(* IEC 61131-3 sources: OpenPLC_Sample_Programs/successed_ST, 85 files *)

(* ---- complex_arithmetic.st ---- *)
FUNCTION_BLOCK SLIDINGMEAN_A
  VAR_INPUT  START, END, VALUE : INT; END_VAR
  VAR MEAN : INT := 0; WEIGHT  : INT := 1; END_VAR
  VAR_OUTPUT Q : INT; END_VAR

  IF START < END THEN
    MEAN := (END - START) / WEIGHT * VALUE + MEAN;
    WEIGHT := END - START + WEIGHT;
  END_IF;
  Q := MEAN;
END_FUNCTION_BLOCK

FUNCTION_BLOCK SLIDINGMEAN_B
  VAR_INPUT  START, END, VALUE : INT;
             RESET : BOOL;
  END_VAR
  VAR MEAN :INT := 0; WEIGHT  : INT := 1; END_VAR
  VAR_OUTPUT Q : INT; END_VAR

  IF RESET THEN
    WEIGHT := 1; MEAN := 0;
  ELSIF START < END THEN
    MEAN := (END - START) * VALUE + WEIGHT * MEAN;
    WEIGHT := END - START + WEIGHT;
  END_IF;

END_FUNCTION_BLOCK

PROGRAM WARN_ABOVE
  VAR SENSOR, THRESHOLD : INT; END_VAR
  VAR SM : SLIDINGMEAN_A; END_VAR
  VAR_OUTPUT CRITICAL : BOOL; END_VAR
  SM(START := 0, END := 7, VALUE := SENSOR);
  CRITICAL :=  SM.Q > THRESHOLD;
END_PROGRAM

PROGRAM WARN_BELOW
  VAR SENSOR, THRESHOLD : INT; END_VAR
  VAR SM : SLIDINGMEAN_A; END_VAR
  VAR_OUTPUT CRITICAL : BOOL; END_VAR
  SM(START := 0, END := 7, VALUE := SENSOR);
  CRITICAL :=  SM.Q <= THRESHOLD;
END_PROGRAM

CONFIGURATION Config0
  RESOURCE Res0 ON PLC
    TASK TASK0(INTERVAL := T#50MS, PRIORITY := 0);
    PROGRAM INSTANCE0 WITH TASK0 : WARN_ABOVE;
    PROGRAM INSTANCE1 WITH TASK0 : WARN_BELOW;
  END_RESOURCE
END_CONFIGURATION

(* ---- fbembedding_1.st ---- *)
FUNCTION_BLOCK FB1

VAR_INPUT J : INT; END_VAR
VAR_OUTPUT P : INT; END_VAR
VAR SUM : INT; END_VAR

SUM := P + SUM;
P := SUM / P;

END_FUNCTION_BLOCK

PROGRAM MAIN
VAR_INPUT I : INT; END_VAR
VAR_OUTPUT O : INT; END_VAR

VAR
   A : FB1;
END_VAR
A(J:=I);
O:=A.P;
END_PROGRAM

CONFIGURATION Config0
  RESOURCE Res0 ON PLC
    TASK TASK0(INTERVAL := T#50MS, PRIORITY := 0);
    PROGRAM INSTANCE0 WITH TASK0 : MAIN;
  END_RESOURCE
END_CONFIGURATION

(* ---- lr.real.st ---- *)
TYPE
  OpMode : (Op , Teach);
  TeachStatus :  (Ok, NoTeachPoints, Teaching, InvalidTeachPoints, InvalidInputValue);
END_TYPE

FUNCTION_BLOCK TON_B

VAR_INPUT
  IN : BOOL;
  PT : INT;
END_VAR

VAR_OUTPUT
  Q  : BOOL;
  ET : INT;
END_VAR

IF IN THEN
  Q:= ET = INT#0;
  IF ET > INT#0 THEN
      ET := ET - INT#1;
  ELSE
      ET := INT#0;
  END_IF;
ELSE
  Q  := FALSE;
  ET := PT;
END_IF;

END_FUNCTION_BLOCK

PROGRAM Analogsensor

VAR
  SENSORINPUT_MIN : REAL := REAL#0.0;
  SENSORINPUT_MAX : REAL := REAL#4095.0;
  TEACHTIMEOUT : TIME := TIME#20s0ms;
END_VAR

VAR_INPUT
  TPSet : BOOL;
  SensorInput, TPy  : INT;
  OperationMode : OpMode;
END_VAR

VAR_OUTPUT
  SensorOutput : INT;
END_VAR

VAR
  initial          : BOOL;
  lastmode         : OpMode;
  Status           : TeachStatus;
  teachstep        : INT;
  x_temp, y_temp, t, m, x1, y1, x2, y2 : REAL;
  timeout          	: TON_B;
END_VAR

IF NOT initial THEN
  x1 := 0.0;
  y1 := 0.0;
  x2 := 0.0;
  y2 := 0.0;
  Status := TeachStatus#NoTeachPoints;
  initial := TRUE;
ELSE
  IF OperationMode = OpMode#Op THEN
    IF Status = TeachStatus#Ok AND INT_TO_REAL(SensorInput) >= SENSORINPUT_MIN AND INT_TO_REAL(SensorInput) <= SENSORINPUT_MAX THEN
      SensorOutput := REAL_TO_INT(m) * SensorInput + REAL_TO_INT(t);
    ELSE
      SensorOutput := 0;
    END_IF;
  ELSIF OperationMode = OpMode#Teach THEN
    IF lastmode <> OperationMode THEN
      teachstep := 0;
      timeout(IN := FALSE);
    END_IF;

    CASE teachstep OF
      0:
         Status := TeachStatus#Teaching;
         timeout(IN := TRUE, PT:=TIME_TO_INT(TEACHTIMEOUT));
         IF timeout.Q THEN
           OperationMode := OpMode#Op;
         END_IF;

         IF TPSet AND INT_TO_REAL(SensorInput) >= SENSORINPUT_MIN AND INT_TO_REAL(SensorInput) <= SENSORINPUT_MAX THEN
           y1 := INT_TO_REAL(TPy);
           x1 := INT_TO_REAL(SensorInput);
           teachstep := 1;
           timeout(IN := FALSE);
         END_IF;
      1:
         IF TPSet = FALSE THEN
           teachstep := 2;
         END_IF;
      2:
         timeout(IN := TRUE, PT:=TIME_TO_INT(TEACHTIMEOUT));

         IF timeout.Q THEN
           OperationMode := OpMode#Op;
         END_IF;

         IF TPSet AND INT_TO_REAL(SensorInput) >= SENSORINPUT_MIN
             AND INT_TO_REAL(SensorInput) <= SENSORINPUT_MAX THEN
           y2 := INT_TO_REAL(TPy);
           x2 := INT_TO_REAL(SensorInput);
           teachstep := 3;
           timeout(IN := FALSE);
         END_IF;
       3:
        IF x1 > x2 THEN
           x_temp := x1;
           y_temp := y1;
           x1 := x2;
           y1 := y2;
           x2 := x_temp;
           y2 := y_temp;
        END_IF;

        IF x2 - x1 <> 0.0 THEN
           m   := (y2 - y1) / (x2 - x1);
           t   := y1 - m * x1;
           Status := TeachStatus#Ok;
        ELSE
           Status := TeachStatus#InvalidTeachPoints;
           OperationMode := OpMode#Op;
         END_IF;
       END_CASE;
  END_IF;
END_IF;
  lastmode := OperationMode;
END_PROGRAM

CONFIGURATION Config0
  RESOURCE Res0 ON PLC
    TASK task0(INTERVAL := T#50ms, PRIORITY := 0);
    PROGRAM instance0 WITH task0 : Analogsensor;
  END_RESOURCE
END_CONFIGURATION

(* ---- PPU_13+ESystem.st ---- *)
(**********************************************************)
(* INCLUDED FROM ESYSTEM.ST                               *)

FUNCTION_BLOCK RS_FF
	VAR_INPUT    R,S : BOOL; END_VAR
	VAR_OUTPUT     Q : BOOL; END_VAR

	IF S THEN
		Q := TRUE;
	END_IF;
	IF R THEN
		Q := FALSE;
	END_IF;
END_FUNCTION_BLOCK

FUNCTION_BLOCK ESYSTEM
    VAR_INPUT RESET, MANUALSTAMPSLIDEROUT, MANUALSTAMPSLIDERIN,
    		    CRANEPRESSUREON,CRANEPRESSUREOFF: BOOL; END_VAR

    VAR_OUTPUT NEWCRANEPRESSURE : INT;
    			STAMPSLIDERIN, STAMPSLIDEROUT: BOOL; END_VAR

    VAR CONSTANT REGULARCRANEPRESSURE : INT := INT#8600; END_VAR

    VAR CRANEPRESSURE : RS_FF := (Q:=TRUE);
    	   RTRIGSTAMPSLIDERIN, RTRIGSTAMPSLIDEROUT : R_TRIG;
    END_VAR

	IF RESET THEN
		CRANEPRESSURE(S:=TRUE,R:=FALSE);
		RTRIGSTAMPSLIDERIN(CLK:=FALSE);
		RTRIGSTAMPSLIDEROUT(CLK:=FALSE);
	END_IF;

	CRANEPRESSURE(S:=CRANEPRESSUREON, R:=CRANEPRESSUREOFF);
	IF CRANEPRESSURE.Q THEN
		NEWCRANEPRESSURE := INT#0;
    	ELSE
    		NEWCRANEPRESSURE := REGULARCRANEPRESSURE;
    	END_IF;

	RTRIGSTAMPSLIDERIN(CLK:=STAMPSLIDERIN);
	RTRIGSTAMPSLIDEROUT(CLK:=STAMPSLIDEROUT);

	IF MANUALSTAMPSLIDEROUT AND RTRIGSTAMPSLIDERIN.Q THEN
		STAMPSLIDERIN := FALSE;
	ELSIF MANUALSTAMPSLIDEROUT THEN
		STAMPSLIDEROUT := TRUE;
	END_IF;

	IF MANUALSTAMPSLIDERIN AND RTRIGSTAMPSLIDEROUT.Q THEN
		STAMPSLIDEROUT := FALSE;
	ELSIF MANUALSTAMPSLIDEROUT THEN
		STAMPSLIDEROUT := TRUE;
	END_IF;
END_FUNCTION_BLOCK
(**********************************************************)

TYPE

    MAGAZIN_STATES_T : (GREEN_LAMP, INIT, INTERSTEP, MAGAZIN_INIT,
    MAGAZIN_INIT_2, SLIDER_MOVE_BACK, START_MAGAZIN, STEP0, STEP1, CONVEY);

    STAMP_STATES_T : (GREEN_LAMP, INIT, INTERSTEP, INTERSTEP_2, STAMPPROCESS,
    STAMPSLIDERBACK, STAMPSLIDERFORWARD, STAMP_INIT_1, STAMP_INIT_2,
    STAMP_INIT_3, STAMP_INIT_4, START_STAMP, STEP0, STEP1, STEP2);

    CRANE_STATES_T : (CRANE_GO_UP, CRANE_INIT, CRANE_INIT_2,
    CRANE_LIFT_AT_STAMP, CRANE_LIFT_CONVEYOR, CRANE_LIFT_CONVEYOR_BLACK,
    CRANE_LIFT_MAGAZIN, CRANE_LIFT_MAGAZIN_METALLIC,
    CRANE_LIFT_NOT_METALLIC_BLACK, CRANE_LOWER, CRANE_ON_CONVEYOR,
    CRANE_ON_CONVEYOR_METALLIC, CRANE_ON_CONVEYOR_NOT_METALLICA_BLACK,
    CRANE_ON_STAMP_METALLIC, CRANE_ON_STAMP_STOP_BLACK,
    CRANE_TURN_LEFT_BACK_TO_STAMP, CRANE_TURN_LEFT_FROM_STAMP,
    CRANE_TURN_LEFT_METALLIC, CRANE_TURN_LEFT_NOT_METALLIC,
    CRANE_TURN_LEFT_NOT_METALLIC_BLACK, INIT, INTERSTEP, INTERSTEP_2,
    LAST_WORKPIECE_AT_STAMP, LOWER_CRANE, MAGAZIN_STOP, MAGAZIN_STOP_BLACK,
    NO_WORKPIECE_READY, RESET_INTERCONNECT, START_CRANE, STEP0, SUCK_AT_STAMP,
    TIMEDELAY, TURN_RIGHT, TURN_RIGHT_BLACK, PAUSE, RELEASE, RELEASE_BLACK,
    RELEASE_WORKPIECE);

END_TYPE

FUNCTION_BLOCK MAGAZIN
    VAR_INPUT  CRANEDOWN : BOOL; END_VAR
    VAR_OUTPUT  CRANELOWER : BOOL; END_VAR
    VAR_INPUT  CRANEONCONVEYOR : BOOL; END_VAR
    VAR_INPUT  CRANEONMAGAZIN : BOOL; END_VAR
    VAR_INPUT  CRANESUCKED : BOOL; END_VAR
    VAR_OUTPUT  CRANETURNCLOCKWISE : BOOL; END_VAR
    VAR_OUTPUT  CRANETURNCOUNTERCLOCKWISE : BOOL; END_VAR
    VAR_INPUT  CRANEUP : BOOL; END_VAR
    VAR_OUTPUT  MAGAZINGREENLAMP : BOOL; END_VAR
    VAR_OUTPUT  MAGAZINSLIDER : BOOL; END_VAR
    VAR_OUTPUT  MAGAZINVACUUMOFF : BOOL; END_VAR
    VAR_OUTPUT  MAGAZINVACUUMON : BOOL; END_VAR
    VAR_OUTPUT  MAGAZINWHITELAMP : BOOL; END_VAR
    VAR  SFCINIT : BOOL; END_VAR
    VAR_INPUT  SFCRESET : BOOL; END_VAR
    VAR_INPUT  SLIDERMOVEDOUT : BOOL; END_VAR
    VAR_INPUT  SLIDERNOTMOVEDOUT : BOOL; END_VAR
    VAR_INPUT  STARTBUTTONMAGAZIN : BOOL; END_VAR
    VAR_OUTPUT  STARTCOMMANDMAGAZIN : BOOL; END_VAR
    VAR_INPUT  STARTVAR : BOOL; END_VAR
    VAR_INPUT  WORKPIECEREADY : BOOL; END_VAR
    VAR  _STATE : MAGAZIN_STATES_T; END_VAR
    VAR  _TRANSIT : BOOL; END_VAR
    VAR  INTERCONNECTMAGAZINSTARTCOMMAND : BOOL; END_VAR

    CASE _STATE OF
        MAGAZIN_STATES_T#GREEN_LAMP:
            _TRANSIT := FALSE;
            MAGAZINGREENLAMP := TRUE;
            INTERCONNECTMAGAZINSTARTCOMMAND := FALSE;
            IF TRUE THEN
                _TRANSIT := TRUE;
                _STATE := MAGAZIN_STATES_T#MAGAZIN_INIT;
            END_IF;

        MAGAZIN_STATES_T#INIT:
            _TRANSIT := FALSE;
            IF TRUE THEN
                _TRANSIT := TRUE;
                _STATE := MAGAZIN_STATES_T#START_MAGAZIN;
            END_IF;

        MAGAZIN_STATES_T#INTERSTEP:
            _TRANSIT := FALSE;
            STARTCOMMANDMAGAZIN := TRUE;
            IF STARTVAR THEN
                _TRANSIT := TRUE;
                _STATE := MAGAZIN_STATES_T#CONVEY;
            END_IF;

        MAGAZIN_STATES_T#MAGAZIN_INIT:
            _TRANSIT := FALSE;
            MAGAZINSLIDER := TRUE;
            IF TRUE THEN
                _TRANSIT := TRUE;
                _STATE := MAGAZIN_STATES_T#MAGAZIN_INIT_2;
            END_IF;

        MAGAZIN_STATES_T#MAGAZIN_INIT_2:
            _TRANSIT := FALSE;
            MAGAZINSLIDER := FALSE;
            IF TRUE THEN
                _TRANSIT := TRUE;
                _STATE := MAGAZIN_STATES_T#INTERSTEP;
            END_IF;

        MAGAZIN_STATES_T#SLIDER_MOVE_BACK:
            _TRANSIT := FALSE;
            IF ((SLIDERMOVEDOUT = TRUE) AND (SLIDERNOTMOVEDOUT = FALSE)) THEN
                MAGAZINSLIDER := FALSE;
            END_IF;
            IF CRANEUP THEN
                _TRANSIT := TRUE;
                _STATE := MAGAZIN_STATES_T#STEP1;
            END_IF;

        MAGAZIN_STATES_T#START_MAGAZIN:
            _TRANSIT := FALSE;
            MAGAZINSLIDER := FALSE;
            MAGAZINGREENLAMP := FALSE;
            STARTVAR := FALSE;
            STARTCOMMANDMAGAZIN := FALSE;
            IF (STARTBUTTONMAGAZIN = TRUE) THEN
                INTERCONNECTMAGAZINSTARTCOMMAND := TRUE;
            END_IF;
            IF INTERCONNECTMAGAZINSTARTCOMMAND THEN
                _TRANSIT := TRUE;
                _STATE := MAGAZIN_STATES_T#GREEN_LAMP;
            END_IF;

        MAGAZIN_STATES_T#STEP0:
            _TRANSIT := FALSE;
            IF CRANEDOWN THEN
                _TRANSIT := TRUE;
                _STATE := MAGAZIN_STATES_T#SLIDER_MOVE_BACK;
            END_IF;

        MAGAZIN_STATES_T#STEP1:
            _TRANSIT := FALSE;
            IF CRANEONCONVEYOR THEN
                _TRANSIT := TRUE;
                _STATE := MAGAZIN_STATES_T#INTERSTEP;
            END_IF;

        MAGAZIN_STATES_T#CONVEY:
            _TRANSIT := FALSE;
            IF SLIDERNOTMOVEDOUT THEN
                MAGAZINSLIDER := TRUE;
            END_IF;
            IF CRANEONMAGAZIN THEN
                _TRANSIT := TRUE;
                _STATE := MAGAZIN_STATES_T#STEP0;
            END_IF;

            END_CASE;
END_FUNCTION_BLOCK

FUNCTION_BLOCK STAMP_FB
VAR_INPUT  CRANEDOWN : BOOL; END_VAR
VAR_INPUT  CRANEONCONVEYOR : BOOL; END_VAR
VAR_INPUT  CRANEPOSITIONSTAMP : BOOL; END_VAR
VAR_INPUT  CRANESUCKED : BOOL; END_VAR
VAR_INPUT  CRANEUP : BOOL; END_VAR
VAR  DURATION : TIME := TIME#500MS; END_VAR
VAR  SFCINIT : BOOL; END_VAR
VAR_INPUT  SFCRESET : BOOL; END_VAR
VAR_OUTPUT  STAMPGREENLAMP : BOOL; END_VAR
VAR_INPUT  STAMPLOWERED : BOOL; END_VAR
VAR_OUTPUT  STAMPPRESSURE : BOOL; END_VAR
VAR_OUTPUT  STAMPPUSHER : BOOL; END_VAR
VAR_INPUT  STAMPSLIDERFILLED : BOOL; END_VAR
VAR_OUTPUT  STAMPSLIDERMOVEDIN : BOOL; END_VAR
VAR_OUTPUT  STAMPSLIDERMOVEDOUT : BOOL; END_VAR
VAR_INPUT  STAMPSLIDERSENSORMOVEDIN : BOOL; END_VAR
VAR_INPUT  STAMPSLIDERSENSORMOVEDOUT : BOOL; END_VAR
VAR_INPUT  STAMPSTARTBUTTON : BOOL; END_VAR
VAR_INPUT  STAMPUP : BOOL; END_VAR
VAR_OUTPUT  STAMPWHITELAMP : BOOL; END_VAR
VAR_OUTPUT  STARTCOMMANDSTAMP : BOOL; END_VAR
VAR_INPUT  STARTVAR : BOOL; END_VAR
VAR  TIMER : TON; END_VAR
VAR  _STATE : STAMP_STATES_T; END_VAR
VAR  _TRANSIT : BOOL; END_VAR
VAR  INTERCONNECT : BOOL; END_VAR
VAR  INTERCONNECTSTAMPSTARTCOMMAND : BOOL; END_VAR

CASE _STATE OF
    STAMP_STATES_T#GREEN_LAMP:
        _TRANSIT := FALSE;
        STAMPGREENLAMP := TRUE;
        INTERCONNECTSTAMPSTARTCOMMAND := FALSE;
        IF TRUE THEN
            _TRANSIT := TRUE;
            _STATE := STAMP_STATES_T#STAMP_INIT_1;
        END_IF;

    STAMP_STATES_T#INIT:
        _TRANSIT := FALSE;
        IF TRUE THEN
            _TRANSIT := TRUE;
            _STATE := STAMP_STATES_T#START_STAMP;
        END_IF;

    STAMP_STATES_T#INTERSTEP:
        _TRANSIT := FALSE;
        STARTCOMMANDSTAMP := TRUE;
        IF STARTVAR THEN
            _TRANSIT := TRUE;
            _STATE := STAMP_STATES_T#INTERSTEP_2;
        END_IF;

    STAMP_STATES_T#INTERSTEP_2:
        _TRANSIT := FALSE;
        IF STAMPSLIDERFILLED THEN
            _TRANSIT := TRUE;
            _STATE := STAMP_STATES_T#STEP0;
        END_IF;

    STAMP_STATES_T#STAMPPROCESS:
        _TRANSIT := FALSE;
        STAMPSLIDERMOVEDIN := FALSE;
        STAMPPUSHER := TRUE;
        IF STAMPLOWERED THEN
            _TRANSIT := TRUE;
            _STATE := STAMP_STATES_T#STEP1;
        END_IF;

    STAMP_STATES_T#STAMPSLIDERBACK:
        _TRANSIT := FALSE;
        STAMPSLIDERMOVEDIN := TRUE;
        STAMPSLIDERMOVEDOUT := FALSE;
        IF STAMPSLIDERSENSORMOVEDIN THEN
            _TRANSIT := TRUE;
            _STATE := STAMP_STATES_T#STAMPPROCESS;
        END_IF;

    STAMP_STATES_T#STAMPSLIDERFORWARD:
        _TRANSIT := FALSE;
        STAMPPUSHER := FALSE;
        STAMPSLIDERMOVEDOUT := TRUE;
        IF ((STAMPLOWERED = FALSE) AND (STAMPUP = TRUE)) THEN
            INTERCONNECT := FALSE;
        END_IF;
        TIMER(IN := FALSE, PT := TIME#1MS);
        IF STAMPSLIDERMOVEDOUT THEN
            _TRANSIT := TRUE;
            _STATE := STAMP_STATES_T#STEP2;
        END_IF;

    STAMP_STATES_T#STAMP_INIT_1:
        _TRANSIT := FALSE;
        STAMPSLIDERMOVEDIN := TRUE;
        STAMPSLIDERMOVEDOUT := FALSE;
        IF STAMPSLIDERSENSORMOVEDIN THEN
            _TRANSIT := TRUE;
            _STATE := STAMP_STATES_T#STAMP_INIT_2;
        END_IF;

    STAMP_STATES_T#STAMP_INIT_2:
        _TRANSIT := FALSE;
        STAMPSLIDERMOVEDIN := FALSE;
        STAMPSLIDERMOVEDOUT := TRUE;
        IF STAMPSLIDERSENSORMOVEDOUT THEN
            _TRANSIT := TRUE;
            _STATE := STAMP_STATES_T#STAMP_INIT_3;
        END_IF;

    STAMP_STATES_T#STAMP_INIT_3:
        _TRANSIT := FALSE;
        STAMPPUSHER := TRUE;
        IF STAMPLOWERED THEN
            _TRANSIT := TRUE;
            _STATE := STAMP_STATES_T#STAMP_INIT_4;
        END_IF;

    STAMP_STATES_T#STAMP_INIT_4:
        _TRANSIT := FALSE;
        STAMPPUSHER := FALSE;
        IF STAMPUP THEN
            _TRANSIT := TRUE;
            _STATE := STAMP_STATES_T#INTERSTEP;
        END_IF;

    STAMP_STATES_T#START_STAMP:
        _TRANSIT := FALSE;
        STAMPSLIDERMOVEDOUT := FALSE;
        STAMPSLIDERMOVEDIN := FALSE;
        STAMPPUSHER := FALSE;
        STAMPGREENLAMP := FALSE;
        STAMPPRESSURE := FALSE;
        STARTCOMMANDSTAMP := FALSE;
        IF (STAMPSTARTBUTTON = TRUE) THEN
            INTERCONNECTSTAMPSTARTCOMMAND := TRUE;
        END_IF;
        IF INTERCONNECTSTAMPSTARTCOMMAND THEN
            _TRANSIT := TRUE;
            _STATE := STAMP_STATES_T#GREEN_LAMP;
        END_IF;

    STAMP_STATES_T#STEP0:
        _TRANSIT := FALSE;
        IF CRANEUP THEN
            _TRANSIT := TRUE;
            _STATE := STAMP_STATES_T#STAMPSLIDERBACK;
        END_IF;

    STAMP_STATES_T#STEP1:
        _TRANSIT := FALSE;
        TIMER(IN := STAMPLOWERED, PT := TIME#12MS);
        INTERCONNECT := TIMER.Q;
        IF INTERCONNECT THEN
            _TRANSIT := TRUE;
            _STATE := STAMP_STATES_T#STAMPSLIDERFORWARD;
        END_IF;

    STAMP_STATES_T#STEP2:
        _TRANSIT := FALSE;
        IF (CRANEONCONVEYOR AND NOT STAMPSLIDERFILLED) THEN
            _TRANSIT := TRUE;
            _STATE := STAMP_STATES_T#INTERSTEP;
        END_IF;

    END_CASE;
END_FUNCTION_BLOCK

FUNCTION_BLOCK CRANE_FB
VAR  CRANTURNCLOCKWISE : BOOL; END_VAR
VAR_INPUT  CRANEDOWN : BOOL; END_VAR
VAR_OUTPUT  CRANELOWER : BOOL; END_VAR
VAR_INPUT  CRANEONCONVEYOR : BOOL; END_VAR
VAR_INPUT  CRANEONMAGAZIN : BOOL; END_VAR
VAR_INPUT  CRANEPOSITIONSTAMP : BOOL; END_VAR
VAR_INPUT  CRANESUCKED : BOOL; END_VAR
VAR_OUTPUT  CRANETURNCLOCKWISE : BOOL; END_VAR
VAR_OUTPUT  CRANETURNCOUNTERCLOCKWISE : BOOL; END_VAR
VAR_INPUT  CRANEUP : BOOL; END_VAR
VAR  DURATION1 : TIME := TIME#1S500MS; END_VAR
VAR_INPUT  MAGAZINCAPACITIVESENSOR : BOOL; END_VAR
VAR_OUTPUT  MAGAZINSLIDER : BOOL; END_VAR
VAR_OUTPUT  MAGAZINVACUUMOFF : BOOL; END_VAR
VAR_OUTPUT  MAGAZINVACUUMON : BOOL; END_VAR
VAR  SFCINIT : BOOL; END_VAR
VAR_INPUT  SFCRESET : BOOL; END_VAR
VAR_INPUT  SLIDERMOVEDOUT : BOOL; END_VAR
VAR_INPUT  SLIDERNOTMOVEDOUT : BOOL; END_VAR
VAR_INPUT  STAMPLOWERED : BOOL; END_VAR
VAR_INPUT  STAMPSLIDERFILLED : BOOL; END_VAR
VAR_INPUT  STARTBUTTONMAGAZIN : BOOL; END_VAR
VAR_OUTPUT  STARTCOMMANDCRANE : BOOL; END_VAR
VAR_INPUT  STARTVAR : BOOL; END_VAR
VAR  TIMEDELAY_TIMER : TON; END_VAR
VAR  TIMEDELAY_TIMER_DURATION : TIME := TIME#50MS; END_VAR
VAR  TIMEDELAY_TIMER_INTERCONNECT : BOOL; END_VAR
VAR  TIMER1 : TON; END_VAR
VAR_INPUT  WORKPIECEREADY : BOOL; END_VAR
VAR  _STATE : CRANE_STATES_T; END_VAR
VAR  _TRANSIT : BOOL; END_VAR
VAR  ACTUALTIME1 : TIME; END_VAR
VAR  INTERCONNECT : BOOL; END_VAR
VAR  INTERCONNECTCRANESTARTCOMMAND : BOOL; END_VAR

CASE _STATE OF
    CRANE_STATES_T#CRANE_GO_UP:
        _TRANSIT := FALSE;
        CRANELOWER := FALSE;
        IF (CRANEUP AND (MAGAZINCAPACITIVESENSOR OR NOT WORKPIECEREADY)) THEN
            _TRANSIT := TRUE;
            _STATE := CRANE_STATES_T#PAUSE;
        ELSIF ((CRANEUP AND NOT MAGAZINCAPACITIVESENSOR) AND WORKPIECEREADY) THEN
            _TRANSIT := TRUE;
            _STATE := CRANE_STATES_T#TURN_RIGHT_BLACK;
        END_IF;

    CRANE_STATES_T#CRANE_INIT:
        _TRANSIT := FALSE;
        CRANELOWER := TRUE;
        INTERCONNECTCRANESTARTCOMMAND := FALSE;
        IF CRANEDOWN THEN
            _TRANSIT := TRUE;
            _STATE := CRANE_STATES_T#CRANE_INIT_2;
        END_IF;

    CRANE_STATES_T#CRANE_INIT_2:
        _TRANSIT := FALSE;
        CRANELOWER := FALSE;
        IF CRANEUP THEN
            _TRANSIT := TRUE;
            _STATE := CRANE_STATES_T#INTERSTEP;
        END_IF;

    CRANE_STATES_T#CRANE_LIFT_AT_STAMP:
        _TRANSIT := FALSE;
        CRANELOWER := FALSE;
        IF CRANEUP THEN
            _TRANSIT := TRUE;
            _STATE := CRANE_STATES_T#CRANE_TURN_LEFT_FROM_STAMP;
        END_IF;

    CRANE_STATES_T#CRANE_LIFT_CONVEYOR:
        _TRANSIT := FALSE;
        CRANELOWER := FALSE;
        IF TRUE THEN
            _TRANSIT := TRUE;
            _STATE := CRANE_STATES_T#INTERSTEP;
        END_IF;

    CRANE_STATES_T#CRANE_LIFT_CONVEYOR_BLACK:
        _TRANSIT := FALSE;
        CRANELOWER := FALSE;
        IF CRANEUP THEN
            _TRANSIT := TRUE;
            _STATE := CRANE_STATES_T#CRANE_TURN_LEFT_BACK_TO_STAMP;
        END_IF;

    CRANE_STATES_T#CRANE_LIFT_MAGAZIN:
        _TRANSIT := FALSE;
        CRANELOWER := FALSE;
        IF CRANEUP THEN
            _TRANSIT := TRUE;
            _STATE := CRANE_STATES_T#CRANE_TURN_LEFT_NOT_METALLIC;
        END_IF;

    CRANE_STATES_T#CRANE_LIFT_MAGAZIN_METALLIC:
        _TRANSIT := FALSE;
        CRANELOWER := FALSE;
        IF CRANEUP THEN
            _TRANSIT := TRUE;
            _STATE := CRANE_STATES_T#CRANE_TURN_LEFT_METALLIC;
        END_IF;

    CRANE_STATES_T#CRANE_LIFT_NOT_METALLIC_BLACK:
        _TRANSIT := FALSE;
        CRANELOWER := FALSE;
        IF CRANEUP THEN
            _TRANSIT := TRUE;
            _STATE := CRANE_STATES_T#CRANE_TURN_LEFT_NOT_METALLIC_BLACK;
        END_IF;

    CRANE_STATES_T#CRANE_LOWER:
        _TRANSIT := FALSE;
        MAGAZINVACUUMON := TRUE;
        MAGAZINVACUUMOFF := FALSE;
        CRANELOWER := TRUE;
        IF CRANESUCKED THEN
            _TRANSIT := TRUE;
            _STATE := CRANE_STATES_T#STEP0;
        END_IF;

    CRANE_STATES_T#CRANE_ON_CONVEYOR:
        _TRANSIT := FALSE;
        CRANETURNCOUNTERCLOCKWISE := FALSE;
        CRANETURNCLOCKWISE := FALSE;
        CRANELOWER := TRUE;
        IF CRANEDOWN THEN
            _TRANSIT := TRUE;
            _STATE := CRANE_STATES_T#RELEASE;
        END_IF;

    CRANE_STATES_T#CRANE_ON_CONVEYOR_METALLIC:
        _TRANSIT := FALSE;
        CRANETURNCOUNTERCLOCKWISE := FALSE;
        CRANETURNCLOCKWISE := FALSE;
        CRANELOWER := TRUE;
        IF CRANEDOWN THEN
            _TRANSIT := TRUE;
            _STATE := CRANE_STATES_T#RELEASE;
        END_IF;

    CRANE_STATES_T#CRANE_ON_CONVEYOR_NOT_METALLICA_BLACK:
        _TRANSIT := FALSE;
        CRANETURNCOUNTERCLOCKWISE := FALSE;
        CRANETURNCLOCKWISE := FALSE;
        CRANELOWER := TRUE;
        IF CRANEDOWN THEN
            _TRANSIT := TRUE;
            _STATE := CRANE_STATES_T#RELEASE_BLACK;
        END_IF;

    CRANE_STATES_T#CRANE_ON_STAMP_METALLIC:
        _TRANSIT := FALSE;
        CRANETURNCOUNTERCLOCKWISE := FALSE;
        CRANETURNCLOCKWISE := FALSE;
        CRANELOWER := TRUE;
        IF CRANEDOWN THEN
            _TRANSIT := TRUE;
            _STATE := CRANE_STATES_T#RELEASE_WORKPIECE;
        END_IF;

    CRANE_STATES_T#CRANE_ON_STAMP_STOP_BLACK:
        _TRANSIT := FALSE;
        CRANETURNCLOCKWISE := FALSE;
        CRANETURNCOUNTERCLOCKWISE := FALSE;
        IF TRUE THEN
            _TRANSIT := TRUE;
            _STATE := CRANE_STATES_T#RESET_INTERCONNECT;
        END_IF;

    CRANE_STATES_T#CRANE_TURN_LEFT_BACK_TO_STAMP:
        _TRANSIT := FALSE;
        CRANETURNCOUNTERCLOCKWISE := TRUE;
        CRANETURNCLOCKWISE := FALSE;
        IF CRANEPOSITIONSTAMP THEN
            _TRANSIT := TRUE;
            _STATE := CRANE_STATES_T#CRANE_ON_STAMP_STOP_BLACK;
        END_IF;

    CRANE_STATES_T#CRANE_TURN_LEFT_FROM_STAMP:
        _TRANSIT := FALSE;
        CRANETURNCLOCKWISE := TRUE;
        CRANETURNCOUNTERCLOCKWISE := FALSE;
        IF CRANEONCONVEYOR THEN
            _TRANSIT := TRUE;
            _STATE := CRANE_STATES_T#CRANE_ON_CONVEYOR_METALLIC;
        END_IF;

    CRANE_STATES_T#CRANE_TURN_LEFT_METALLIC:
        _TRANSIT := FALSE;
        CRANETURNCOUNTERCLOCKWISE := TRUE;
        CRANETURNCLOCKWISE := FALSE;
        IF CRANEPOSITIONSTAMP THEN
            _TRANSIT := TRUE;
            _STATE := CRANE_STATES_T#CRANE_ON_STAMP_METALLIC;
        END_IF;

    CRANE_STATES_T#CRANE_TURN_LEFT_NOT_METALLIC:
        _TRANSIT := FALSE;
        CRANETURNCOUNTERCLOCKWISE := TRUE;
        CRANETURNCLOCKWISE := FALSE;
        IF CRANEONCONVEYOR THEN
            _TRANSIT := TRUE;
            _STATE := CRANE_STATES_T#CRANE_ON_CONVEYOR;
        END_IF;

    CRANE_STATES_T#CRANE_TURN_LEFT_NOT_METALLIC_BLACK:
        _TRANSIT := FALSE;
        CRANETURNCOUNTERCLOCKWISE := TRUE;
        CRANETURNCLOCKWISE := FALSE;
        IF CRANEONCONVEYOR THEN
            _TRANSIT := TRUE;
            _STATE := CRANE_STATES_T#CRANE_ON_CONVEYOR_NOT_METALLICA_BLACK;
        END_IF;

    CRANE_STATES_T#INIT:
        _TRANSIT := FALSE;
        IF TRUE THEN
            _TRANSIT := TRUE;
            _STATE := CRANE_STATES_T#START_CRANE;
        END_IF;

    CRANE_STATES_T#INTERSTEP:
        _TRANSIT := FALSE;
        STARTCOMMANDCRANE := TRUE;
        IF STARTVAR THEN
            _TRANSIT := TRUE;
            _STATE := CRANE_STATES_T#INTERSTEP_2;
        END_IF;

    CRANE_STATES_T#INTERSTEP_2:
        _TRANSIT := FALSE;
        IF SLIDERMOVEDOUT THEN
            _TRANSIT := TRUE;
            _STATE := CRANE_STATES_T#TIMEDELAY;
        END_IF;

    CRANE_STATES_T#LAST_WORKPIECE_AT_STAMP:
        _TRANSIT := FALSE;
        IF TRUE THEN
            _TRANSIT := TRUE;
            _STATE := CRANE_STATES_T#PAUSE;
        END_IF;

    CRANE_STATES_T#LOWER_CRANE:
        _TRANSIT := FALSE;
        CRANELOWER := TRUE;
        IF CRANEDOWN THEN
            _TRANSIT := TRUE;
            _STATE := CRANE_STATES_T#SUCK_AT_STAMP;
        END_IF;

    CRANE_STATES_T#MAGAZIN_STOP:
        _TRANSIT := FALSE;
        CRANETURNCLOCKWISE := FALSE;
        CRANETURNCOUNTERCLOCKWISE := FALSE;
        IF (NOT WORKPIECEREADY AND NOT STAMPSLIDERFILLED) THEN
            _TRANSIT := TRUE;
            _STATE := CRANE_STATES_T#NO_WORKPIECE_READY;
        ELSIF WORKPIECEREADY THEN
            _TRANSIT := TRUE;
            _STATE := CRANE_STATES_T#CRANE_LOWER;
        ELSIF (NOT WORKPIECEREADY AND STAMPSLIDERFILLED) THEN
            _TRANSIT := TRUE;
            _STATE := CRANE_STATES_T#LAST_WORKPIECE_AT_STAMP;
        END_IF;

    CRANE_STATES_T#MAGAZIN_STOP_BLACK:
        _TRANSIT := FALSE;
        CRANETURNCLOCKWISE := FALSE;
        CRANETURNCOUNTERCLOCKWISE := FALSE;
        MAGAZINVACUUMON := TRUE;
        MAGAZINVACUUMOFF := FALSE;
        CRANELOWER := TRUE;
        IF CRANESUCKED THEN
            _TRANSIT := TRUE;
            _STATE := CRANE_STATES_T#CRANE_LIFT_NOT_METALLIC_BLACK;
        END_IF;

    CRANE_STATES_T#NO_WORKPIECE_READY:
        _TRANSIT := FALSE;
        IF TRUE THEN
            _TRANSIT := TRUE;
            _STATE := CRANE_STATES_T#START_CRANE;
        END_IF;

    CRANE_STATES_T#RESET_INTERCONNECT:
        _TRANSIT := FALSE;
        INTERCONNECT := FALSE;
        TIMER1(IN := FALSE, PT := TIME#1MS);
        IF SLIDERMOVEDOUT THEN
            _TRANSIT := TRUE;
            _STATE := CRANE_STATES_T#LOWER_CRANE;
        END_IF;

    CRANE_STATES_T#START_CRANE:
        _TRANSIT := FALSE;
        CRANELOWER := FALSE;
        MAGAZINVACUUMOFF := TRUE;
        MAGAZINVACUUMON := FALSE;
        CRANETURNCOUNTERCLOCKWISE := FALSE;
        CRANETURNCLOCKWISE := FALSE;
        STARTVAR := FALSE;
        STARTCOMMANDCRANE := FALSE;
        IF (STARTBUTTONMAGAZIN = TRUE) THEN
            INTERCONNECTCRANESTARTCOMMAND := TRUE;
        END_IF;
        IF INTERCONNECTCRANESTARTCOMMAND THEN
            _TRANSIT := TRUE;
            _STATE := CRANE_STATES_T#CRANE_INIT;
        END_IF;

    CRANE_STATES_T#STEP0:
        _TRANSIT := FALSE;
        IF NOT MAGAZINCAPACITIVESENSOR THEN
            _TRANSIT := TRUE;
            _STATE := CRANE_STATES_T#CRANE_LIFT_MAGAZIN;
        ELSIF MAGAZINCAPACITIVESENSOR THEN
            _TRANSIT := TRUE;
            _STATE := CRANE_STATES_T#CRANE_LIFT_MAGAZIN_METALLIC;
        END_IF;

    CRANE_STATES_T#SUCK_AT_STAMP:
        _TRANSIT := FALSE;
        MAGAZINVACUUMON := TRUE;
        MAGAZINVACUUMOFF := FALSE;
        IF CRANESUCKED THEN
            _TRANSIT := TRUE;
            _STATE := CRANE_STATES_T#CRANE_LIFT_AT_STAMP;
        END_IF;

    CRANE_STATES_T#TIMEDELAY:
        _TRANSIT := FALSE;
        TIMEDELAY_TIMER(IN := TRUE, PT := TIMEDELAY_TIMER_DURATION);
        TIMEDELAY_TIMER_INTERCONNECT := TIMEDELAY_TIMER.Q;
        IF TIMEDELAY_TIMER_INTERCONNECT THEN
            _TRANSIT := TRUE;
            _STATE := CRANE_STATES_T#TURN_RIGHT;
        END_IF;

    CRANE_STATES_T#TURN_RIGHT:
        _TRANSIT := FALSE;
        CRANETURNCLOCKWISE := TRUE;
        CRANETURNCOUNTERCLOCKWISE := FALSE;
        IF CRANEONMAGAZIN THEN
            _TRANSIT := TRUE;
            _STATE := CRANE_STATES_T#MAGAZIN_STOP;
        END_IF;

    CRANE_STATES_T#TURN_RIGHT_BLACK:
        _TRANSIT := FALSE;
        CRANETURNCLOCKWISE := TRUE;
        CRANETURNCOUNTERCLOCKWISE := FALSE;
        IF CRANEONMAGAZIN THEN
            _TRANSIT := TRUE;
            _STATE := CRANE_STATES_T#MAGAZIN_STOP_BLACK;
        END_IF;

    CRANE_STATES_T#PAUSE:
        _TRANSIT := FALSE;
        TIMER1(IN := CRANEUP, PT := DURATION1);
        INTERCONNECT := TIMER1.Q;
        IF INTERCONNECT THEN
            _TRANSIT := TRUE;
            _STATE := CRANE_STATES_T#RESET_INTERCONNECT;
        END_IF;

    CRANE_STATES_T#RELEASE:
        _TRANSIT := FALSE;
        MAGAZINVACUUMOFF := TRUE;
        MAGAZINVACUUMON := FALSE;
        IF TRUE THEN
            _TRANSIT := TRUE;
            _STATE := CRANE_STATES_T#CRANE_LIFT_CONVEYOR;
        END_IF;

    CRANE_STATES_T#RELEASE_BLACK:
        _TRANSIT := FALSE;
        MAGAZINVACUUMON := FALSE;
        MAGAZINVACUUMOFF := TRUE;
        IF TRUE THEN
            _TRANSIT := TRUE;
            _STATE := CRANE_STATES_T#CRANE_LIFT_CONVEYOR_BLACK;
        END_IF;

    CRANE_STATES_T#RELEASE_WORKPIECE:
        _TRANSIT := FALSE;
        MAGAZINVACUUMOFF := TRUE;
        MAGAZINVACUUMON := FALSE;
        IF TRUE THEN
            _TRANSIT := TRUE;
            _STATE := CRANE_STATES_T#CRANE_GO_UP;
        END_IF;

    END_CASE;
END_FUNCTION_BLOCK

PROGRAM MAIN

        (** NEW VARIABLES **)
	VAR EMERGENCY : ESYSTEM; END_VAR
	VAR_INPUT
	    SENSOR_MANUALSTAMPSLIDEROUT, SENSOR_MANUALSTAMPSLIDERIN,
	    SENSOR_CRANEPRESSUREON, SENSOR_CRANEPRESSUREOFF : BOOL;
	END_VAR

VAR  CRANE : CRANE_FB; END_VAR
VAR  MAG : MAGAZIN; END_VAR

VAR_OUTPUT ACTUATOR_ANALOGCRANEPRESSURE : INT; END_VAR
VAR_OUTPUT ACTUATOR_CRANELOWER : BOOL; END_VAR
VAR_OUTPUT ACTUATOR_CRANETURNCLOCKWISE : BOOL; END_VAR
VAR_OUTPUT ACTUATOR_CRANETURNCOUNTERCLOCKWISE : BOOL; END_VAR
VAR_OUTPUT ACTUATOR_MAGAZINGREENLAMP : BOOL; END_VAR
VAR_OUTPUT ACTUATOR_MAGAZINSLIDER : BOOL; END_VAR
VAR_OUTPUT ACTUATOR_MAGAZINVACUUMOFF : BOOL; END_VAR
VAR_OUTPUT ACTUATOR_MAGAZINVACUUMON : BOOL; END_VAR
VAR_OUTPUT ACTUATOR_MAGAZINWHITELAMP : BOOL; END_VAR
VAR_OUTPUT ACTUATOR_STAMPGREENLAMP : BOOL; END_VAR
VAR_OUTPUT ACTUATOR_STAMPPUSHER : BOOL; END_VAR
VAR_OUTPUT ACTUATOR_STAMPSLIDERMOVEDIN : BOOL; END_VAR
VAR_OUTPUT ACTUATOR_STAMPSLIDERMOVEDOUT : BOOL; END_VAR
VAR_OUTPUT ACTUATOR_STAMPWHITELAMP : BOOL; END_VAR
VAR_INPUT SENSOR_CRANEDOWN : BOOL; END_VAR
VAR_INPUT SENSOR_CRANEONCONVEYOR : BOOL; END_VAR
VAR_INPUT SENSOR_CRANEONMAGAZIN : BOOL; END_VAR
VAR_INPUT SENSOR_CRANEPOSITION : BOOL; END_VAR
VAR_INPUT SENSOR_CRANEPOSITIONSTAMP : BOOL; END_VAR
VAR_INPUT SENSOR_CRANESUCKED : BOOL; END_VAR
VAR_INPUT SENSOR_CRANEUP : BOOL; END_VAR
VAR_INPUT SENSOR_MAGAZINCAPACITIVESENSOR : BOOL; END_VAR
VAR_INPUT SENSOR_MAGAZINEMERGENCYSTOP : BOOL; END_VAR
VAR_INPUT SENSOR_MAGAZINOPTICALSENSOR : BOOL; END_VAR
VAR_INPUT SENSOR_MAGAZINSWITCHMANUELLAUTOMATIC : BOOL; END_VAR
VAR_INPUT SENSOR_SLIDERMOVEDOUT : BOOL; END_VAR
VAR_INPUT SENSOR_SLIDERNOTMOVEDOUT : BOOL; END_VAR
VAR_INPUT SENSOR_STAMPEMERGENCYSTOP : BOOL; END_VAR
VAR_INPUT SENSOR_STAMPLOWERED : BOOL; END_VAR
VAR_INPUT SENSOR_STAMPSLIDERFILLED : BOOL; END_VAR
VAR_INPUT SENSOR_STAMPSLIDERSENSORMOVEDIN : BOOL; END_VAR
VAR_INPUT SENSOR_STAMPSLIDERSENSORMOVEDOUT : BOOL; END_VAR
VAR_INPUT SENSOR_STAMPSTARTBUTTON : BOOL; END_VAR
VAR_INPUT SENSOR_STAMPSWITCHMANUELLAUTOMATIC : BOOL; END_VAR
VAR_INPUT SENSOR_STAMPUP : BOOL; END_VAR
VAR_INPUT SENSOR_STARTBUTTONMAGAZIN : BOOL; END_VAR
VAR_INPUT SENSOR_WORKPIECEREADY : BOOL; END_VAR
VAR  STAMP : STAMP_FB; END_VAR

CRANE.CRANEDOWN := SENSOR_CRANEDOWN;
CRANE.CRANEONCONVEYOR := SENSOR_CRANEONCONVEYOR;
CRANE.CRANEONMAGAZIN := SENSOR_CRANEONMAGAZIN;
CRANE.CRANEPOSITIONSTAMP := SENSOR_CRANEPOSITIONSTAMP;
CRANE.CRANESUCKED := SENSOR_CRANESUCKED;
CRANE.CRANEUP := SENSOR_CRANEUP;
CRANE.MAGAZINCAPACITIVESENSOR := SENSOR_MAGAZINCAPACITIVESENSOR;
CRANE.SLIDERMOVEDOUT := SENSOR_SLIDERMOVEDOUT;
CRANE.STAMPSLIDERFILLED := SENSOR_STAMPSLIDERFILLED;
CRANE.STARTBUTTONMAGAZIN := SENSOR_STARTBUTTONMAGAZIN;
CRANE.WORKPIECEREADY := SENSOR_WORKPIECEREADY;
MAG.CRANEDOWN := SENSOR_CRANEDOWN;
MAG.CRANEONCONVEYOR := SENSOR_CRANEONCONVEYOR;
MAG.CRANEONMAGAZIN := SENSOR_CRANEONMAGAZIN;
MAG.CRANEUP := SENSOR_CRANEUP;
MAG.SLIDERMOVEDOUT := SENSOR_SLIDERMOVEDOUT;
MAG.SLIDERNOTMOVEDOUT := SENSOR_SLIDERNOTMOVEDOUT;
MAG.STARTBUTTONMAGAZIN := SENSOR_STARTBUTTONMAGAZIN;
MAG.WORKPIECEREADY := SENSOR_WORKPIECEREADY;
STAMP.CRANEDOWN := SENSOR_CRANEDOWN;
STAMP.CRANEONCONVEYOR := SENSOR_CRANEONCONVEYOR;
STAMP.CRANEPOSITIONSTAMP := SENSOR_CRANEPOSITIONSTAMP;
STAMP.CRANESUCKED := SENSOR_CRANESUCKED;
STAMP.CRANEUP := SENSOR_CRANEUP;
STAMP.STAMPLOWERED := SENSOR_STAMPLOWERED;
STAMP.STAMPSLIDERFILLED := SENSOR_STAMPSLIDERFILLED;
STAMP.STAMPSLIDERSENSORMOVEDIN := SENSOR_STAMPSLIDERSENSORMOVEDIN;
STAMP.STAMPSLIDERSENSORMOVEDOUT := SENSOR_STAMPSLIDERSENSORMOVEDOUT;
STAMP.STAMPSTARTBUTTON := SENSOR_STAMPSTARTBUTTON;
STAMP.STAMPUP := SENSOR_STAMPUP;

IF (SENSOR_STAMPEMERGENCYSTOP AND SENSOR_MAGAZINEMERGENCYSTOP) THEN
    MAG();
    CRANE();
    STAMP();
    IF (ACTUATOR_MAGAZINGREENLAMP AND ACTUATOR_STAMPGREENLAMP) THEN
        IF ((STAMP.STARTCOMMANDSTAMP AND CRANE.STARTCOMMANDCRANE) AND MAG.STARTCOMMANDMAGAZIN) THEN
            CRANE.STARTVAR := TRUE;
            MAG.STARTVAR := TRUE;
            STAMP.STARTVAR := TRUE;
        END_IF;
    END_IF;
    CRANE.SFCRESET := FALSE;
    MAG.SFCRESET := FALSE;
    STAMP.SFCRESET := FALSE;
    EMERGENCY.RESET := TRUE;
    EMERGENCY();

    ACTUATOR_ANALOGCRANEPRESSURE := INT#6000;
    ACTUATOR_CRANELOWER := CRANE.CRANELOWER;
    ACTUATOR_CRANETURNCLOCKWISE := CRANE.CRANETURNCLOCKWISE;
    ACTUATOR_CRANETURNCOUNTERCLOCKWISE := CRANE.CRANETURNCOUNTERCLOCKWISE;
    ACTUATOR_MAGAZINGREENLAMP := MAG.MAGAZINGREENLAMP;
    ACTUATOR_MAGAZINSLIDER := MAG.MAGAZINSLIDER;
    ACTUATOR_MAGAZINVACUUMOFF := CRANE.MAGAZINVACUUMOFF;
    ACTUATOR_MAGAZINVACUUMON := CRANE.MAGAZINVACUUMON;
    ACTUATOR_STAMPGREENLAMP := STAMP.STAMPGREENLAMP;
    ACTUATOR_STAMPPUSHER := STAMP.STAMPPUSHER;
    ACTUATOR_STAMPSLIDERMOVEDIN := STAMP.STAMPSLIDERMOVEDIN;
    ACTUATOR_STAMPSLIDERMOVEDOUT := STAMP.STAMPSLIDERMOVEDOUT;
    ACTUATOR_STAMPWHITELAMP := STAMP.STAMPWHITELAMP;

ELSIF (NOT SENSOR_STAMPEMERGENCYSTOP OR NOT SENSOR_MAGAZINEMERGENCYSTOP) THEN
	    (* CALL OF THE NEW EMERGENCY SUBSYSTEM *)
	    EMERGENCY(RESET := FALSE,
	              MANUALSTAMPSLIDEROUT :=  SENSOR_MANUALSTAMPSLIDEROUT,
	              MANUALSTAMPSLIDERIN  := SENSOR_MANUALSTAMPSLIDERIN,
			    CRANEPRESSUREON      := SENSOR_CRANEPRESSUREON,
			    CRANEPRESSUREOFF     := SENSOR_CRANEPRESSUREOFF);

	    ACTUATOR_ANALOGCRANEPRESSURE := EMERGENCY.NEWCRANEPRESSURE;
	    ACTUATOR_STAMPSLIDERMOVEDOUT := EMERGENCY.STAMPSLIDERIN;
	    ACTUATOR_STAMPSLIDERMOVEDIN  := EMERGENCY.STAMPSLIDEROUT;
	    (*/END*)

    ACTUATOR_MAGAZINSLIDER := FALSE;
    ACTUATOR_CRANELOWER := FALSE;
    ACTUATOR_MAGAZINVACUUMON := FALSE;
    ACTUATOR_MAGAZINVACUUMOFF := TRUE;
    ACTUATOR_MAGAZINGREENLAMP := FALSE;
    ACTUATOR_CRANETURNCOUNTERCLOCKWISE := FALSE;
    ACTUATOR_CRANETURNCLOCKWISE := FALSE;
    ACTUATOR_STAMPGREENLAMP := FALSE;
    ACTUATOR_STAMPPUSHER := FALSE;
    CRANE.SFCRESET := TRUE;
    MAG.SFCRESET := TRUE;
    STAMP.SFCRESET := TRUE;
    CRANE.STARTVAR := FALSE;
    MAG.STARTVAR := FALSE;
    STAMP.STARTVAR := FALSE;
END_IF;

END_PROGRAM

CONFIGURATION Config0
  RESOURCE Res0 ON PLC
    TASK TASK0(INTERVAL := T#50MS, PRIORITY := 0);
    PROGRAM INSTANCE0 WITH TASK0 : MAIN;
  END_RESOURCE
END_CONFIGURATION

(* ---- PPU_13.st ---- *)
TYPE

    MAGAZIN_STATES_T : (GREEN_LAMP, INIT, INTERSTEP, MAGAZIN_INIT,
    MAGAZIN_INIT_2, SLIDER_MOVE_BACK, START_MAGAZIN, STEP0, STEP1, CONVEY);

    STAMP_STATES_T : (GREEN_LAMP, INIT, INTERSTEP, INTERSTEP_2, STAMPPROCESS,
    STAMPSLIDERBACK, STAMPSLIDERFORWARD, STAMP_INIT_1, STAMP_INIT_2,
    STAMP_INIT_3, STAMP_INIT_4, START_STAMP, STEP0, STEP1, STEP2);

    CRANE_STATES_T : (CRANE_GO_UP, CRANE_INIT, CRANE_INIT_2,
    CRANE_LIFT_AT_STAMP, CRANE_LIFT_CONVEYOR, CRANE_LIFT_CONVEYOR_BLACK,
    CRANE_LIFT_MAGAZIN, CRANE_LIFT_MAGAZIN_METALLIC,
    CRANE_LIFT_NOT_METALLIC_BLACK, CRANE_LOWER, CRANE_ON_CONVEYOR,
    CRANE_ON_CONVEYOR_METALLIC, CRANE_ON_CONVEYOR_NOT_METALLICA_BLACK,
    CRANE_ON_STAMP_METALLIC, CRANE_ON_STAMP_STOP_BLACK,
    CRANE_TURN_LEFT_BACK_TO_STAMP, CRANE_TURN_LEFT_FROM_STAMP,
    CRANE_TURN_LEFT_METALLIC, CRANE_TURN_LEFT_NOT_METALLIC,
    CRANE_TURN_LEFT_NOT_METALLIC_BLACK, INIT, INTERSTEP, INTERSTEP_2,
    LAST_WORKPIECE_AT_STAMP, LOWER_CRANE, MAGAZIN_STOP, MAGAZIN_STOP_BLACK,
    NO_WORKPIECE_READY, RESET_INTERCONNECT, START_CRANE, STEP0, SUCK_AT_STAMP,
    TIMEDELAY, TURN_RIGHT, TURN_RIGHT_BLACK, PAUSE, RELEASE, RELEASE_BLACK,
    RELEASE_WORKPIECE);

END_TYPE

FUNCTION_BLOCK MAGAZIN
    VAR_INPUT  CRANEDOWN : BOOL; END_VAR
    VAR_OUTPUT  CRANELOWER : BOOL; END_VAR
    VAR_INPUT  CRANEONCONVEYOR : BOOL; END_VAR
    VAR_INPUT  CRANEONMAGAZIN : BOOL; END_VAR
    VAR_INPUT  CRANESUCKED : BOOL; END_VAR
    VAR_OUTPUT  CRANETURNCLOCKWISE : BOOL; END_VAR
    VAR_OUTPUT  CRANETURNCOUNTERCLOCKWISE : BOOL; END_VAR
    VAR_INPUT  CRANEUP : BOOL; END_VAR
    VAR_OUTPUT  MAGAZINGREENLAMP : BOOL; END_VAR
    VAR_OUTPUT  MAGAZINSLIDER : BOOL; END_VAR
    VAR_OUTPUT  MAGAZINVACUUMOFF : BOOL; END_VAR
    VAR_OUTPUT  MAGAZINVACUUMON : BOOL; END_VAR
    VAR_OUTPUT  MAGAZINWHITELAMP : BOOL; END_VAR
    VAR  SFCINIT : BOOL; END_VAR
    VAR_INPUT  SFCRESET : BOOL; END_VAR
    VAR_INPUT  SLIDERMOVEDOUT : BOOL; END_VAR
    VAR_INPUT  SLIDERNOTMOVEDOUT : BOOL; END_VAR
    VAR_INPUT  STARTBUTTONMAGAZIN : BOOL; END_VAR
    VAR_OUTPUT  STARTCOMMANDMAGAZIN : BOOL; END_VAR
    VAR_INPUT  STARTVAR : BOOL; END_VAR
    VAR_INPUT  WORKPIECEREADY : BOOL; END_VAR
    VAR  _STATE : MAGAZIN_STATES_T; END_VAR
    VAR  _TRANSIT : BOOL; END_VAR
    VAR  INTERCONNECTMAGAZINSTARTCOMMAND : BOOL; END_VAR

    CASE _STATE OF
        MAGAZIN_STATES_T#GREEN_LAMP:
            _TRANSIT := FALSE;
            MAGAZINGREENLAMP := TRUE;
            INTERCONNECTMAGAZINSTARTCOMMAND := FALSE;
            IF TRUE THEN
                _TRANSIT := TRUE;
                _STATE := MAGAZIN_STATES_T#MAGAZIN_INIT;
            END_IF;

        MAGAZIN_STATES_T#INIT:
            _TRANSIT := FALSE;
            IF TRUE THEN
                _TRANSIT := TRUE;
                _STATE := MAGAZIN_STATES_T#START_MAGAZIN;
            END_IF;

        MAGAZIN_STATES_T#INTERSTEP:
            _TRANSIT := FALSE;
            STARTCOMMANDMAGAZIN := TRUE;
            IF STARTVAR THEN
                _TRANSIT := TRUE;
                _STATE := MAGAZIN_STATES_T#CONVEY;
            END_IF;

        MAGAZIN_STATES_T#MAGAZIN_INIT:
            _TRANSIT := FALSE;
            MAGAZINSLIDER := TRUE;
            IF TRUE THEN
                _TRANSIT := TRUE;
                _STATE := MAGAZIN_STATES_T#MAGAZIN_INIT_2;
            END_IF;

        MAGAZIN_STATES_T#MAGAZIN_INIT_2:
            _TRANSIT := FALSE;
            MAGAZINSLIDER := FALSE;
            IF TRUE THEN
                _TRANSIT := TRUE;
                _STATE := MAGAZIN_STATES_T#INTERSTEP;
            END_IF;

        MAGAZIN_STATES_T#SLIDER_MOVE_BACK:
            _TRANSIT := FALSE;
            IF ((SLIDERMOVEDOUT = TRUE) AND (SLIDERNOTMOVEDOUT = FALSE)) THEN
                MAGAZINSLIDER := FALSE;
            END_IF;
            IF CRANEUP THEN
                _TRANSIT := TRUE;
                _STATE := MAGAZIN_STATES_T#STEP1;
            END_IF;

        MAGAZIN_STATES_T#START_MAGAZIN:
            _TRANSIT := FALSE;
            MAGAZINSLIDER := FALSE;
            MAGAZINGREENLAMP := FALSE;
            STARTVAR := FALSE;
            STARTCOMMANDMAGAZIN := FALSE;
            IF (STARTBUTTONMAGAZIN = TRUE) THEN
                INTERCONNECTMAGAZINSTARTCOMMAND := TRUE;
            END_IF;
            IF INTERCONNECTMAGAZINSTARTCOMMAND THEN
                _TRANSIT := TRUE;
                _STATE := MAGAZIN_STATES_T#GREEN_LAMP;
            END_IF;

        MAGAZIN_STATES_T#STEP0:
            _TRANSIT := FALSE;
            IF CRANEDOWN THEN
                _TRANSIT := TRUE;
                _STATE := MAGAZIN_STATES_T#SLIDER_MOVE_BACK;
            END_IF;

        MAGAZIN_STATES_T#STEP1:
            _TRANSIT := FALSE;
            IF CRANEONCONVEYOR THEN
                _TRANSIT := TRUE;
                _STATE := MAGAZIN_STATES_T#INTERSTEP;
            END_IF;

        MAGAZIN_STATES_T#CONVEY:
            _TRANSIT := FALSE;
            IF SLIDERNOTMOVEDOUT THEN
                MAGAZINSLIDER := TRUE;
            END_IF;
            IF CRANEONMAGAZIN THEN
                _TRANSIT := TRUE;
                _STATE := MAGAZIN_STATES_T#STEP0;
            END_IF;

            END_CASE;
END_FUNCTION_BLOCK

FUNCTION_BLOCK STAMP_FB
VAR_INPUT  CRANEDOWN : BOOL; END_VAR
VAR_INPUT  CRANEONCONVEYOR : BOOL; END_VAR
VAR_INPUT  CRANEPOSITIONSTAMP : BOOL; END_VAR
VAR_INPUT  CRANESUCKED : BOOL; END_VAR
VAR_INPUT  CRANEUP : BOOL; END_VAR
VAR  DURATION : TIME := TIME#500MS; END_VAR
VAR  SFCINIT : BOOL; END_VAR
VAR_INPUT  SFCRESET : BOOL; END_VAR
VAR_OUTPUT  STAMPGREENLAMP : BOOL; END_VAR
VAR_INPUT  STAMPLOWERED : BOOL; END_VAR
VAR_OUTPUT  STAMPPRESSURE : BOOL; END_VAR
VAR_OUTPUT  STAMPPUSHER : BOOL; END_VAR
VAR_INPUT  STAMPSLIDERFILLED : BOOL; END_VAR
VAR_OUTPUT  STAMPSLIDERMOVEDIN : BOOL; END_VAR
VAR_OUTPUT  STAMPSLIDERMOVEDOUT : BOOL; END_VAR
VAR_INPUT  STAMPSLIDERSENSORMOVEDIN : BOOL; END_VAR
VAR_INPUT  STAMPSLIDERSENSORMOVEDOUT : BOOL; END_VAR
VAR_INPUT  STAMPSTARTBUTTON : BOOL; END_VAR
VAR_INPUT  STAMPUP : BOOL; END_VAR
VAR_OUTPUT  STAMPWHITELAMP : BOOL; END_VAR
VAR_OUTPUT  STARTCOMMANDSTAMP : BOOL; END_VAR
VAR_INPUT  STARTVAR : BOOL; END_VAR
VAR  TIMER : TON; END_VAR
VAR  _STATE : STAMP_STATES_T; END_VAR
VAR  _TRANSIT : BOOL; END_VAR
VAR  INTERCONNECT : BOOL; END_VAR
VAR  INTERCONNECTSTAMPSTARTCOMMAND : BOOL; END_VAR

CASE _STATE OF
    STAMP_STATES_T#GREEN_LAMP:
        _TRANSIT := FALSE;
        STAMPGREENLAMP := TRUE;
        INTERCONNECTSTAMPSTARTCOMMAND := FALSE;
        IF TRUE THEN
            _TRANSIT := TRUE;
            _STATE := STAMP_STATES_T#STAMP_INIT_1;
        END_IF;

    STAMP_STATES_T#INIT:
        _TRANSIT := FALSE;
        IF TRUE THEN
            _TRANSIT := TRUE;
            _STATE := STAMP_STATES_T#START_STAMP;
        END_IF;

    STAMP_STATES_T#INTERSTEP:
        _TRANSIT := FALSE;
        STARTCOMMANDSTAMP := TRUE;
        IF STARTVAR THEN
            _TRANSIT := TRUE;
            _STATE := STAMP_STATES_T#INTERSTEP_2;
        END_IF;

    STAMP_STATES_T#INTERSTEP_2:
        _TRANSIT := FALSE;
        IF STAMPSLIDERFILLED THEN
            _TRANSIT := TRUE;
            _STATE := STAMP_STATES_T#STEP0;
        END_IF;

    STAMP_STATES_T#STAMPPROCESS:
        _TRANSIT := FALSE;
        STAMPSLIDERMOVEDIN := FALSE;
        STAMPPUSHER := TRUE;
        IF STAMPLOWERED THEN
            _TRANSIT := TRUE;
            _STATE := STAMP_STATES_T#STEP1;
        END_IF;

    STAMP_STATES_T#STAMPSLIDERBACK:
        _TRANSIT := FALSE;
        STAMPSLIDERMOVEDIN := TRUE;
        STAMPSLIDERMOVEDOUT := FALSE;
        IF STAMPSLIDERSENSORMOVEDIN THEN
            _TRANSIT := TRUE;
            _STATE := STAMP_STATES_T#STAMPPROCESS;
        END_IF;

    STAMP_STATES_T#STAMPSLIDERFORWARD:
        _TRANSIT := FALSE;
        STAMPPUSHER := FALSE;
        STAMPSLIDERMOVEDOUT := TRUE;
        IF ((STAMPLOWERED = FALSE) AND (STAMPUP = TRUE)) THEN
            INTERCONNECT := FALSE;
        END_IF;
        TIMER(IN := FALSE, PT := TIME#1MS);
        IF STAMPSLIDERMOVEDOUT THEN
            _TRANSIT := TRUE;
            _STATE := STAMP_STATES_T#STEP2;
        END_IF;

    STAMP_STATES_T#STAMP_INIT_1:
        _TRANSIT := FALSE;
        STAMPSLIDERMOVEDIN := TRUE;
        STAMPSLIDERMOVEDOUT := FALSE;
        IF STAMPSLIDERSENSORMOVEDIN THEN
            _TRANSIT := TRUE;
            _STATE := STAMP_STATES_T#STAMP_INIT_2;
        END_IF;

    STAMP_STATES_T#STAMP_INIT_2:
        _TRANSIT := FALSE;
        STAMPSLIDERMOVEDIN := FALSE;
        STAMPSLIDERMOVEDOUT := TRUE;
        IF STAMPSLIDERSENSORMOVEDOUT THEN
            _TRANSIT := TRUE;
            _STATE := STAMP_STATES_T#STAMP_INIT_3;
        END_IF;

    STAMP_STATES_T#STAMP_INIT_3:
        _TRANSIT := FALSE;
        STAMPPUSHER := TRUE;
        IF STAMPLOWERED THEN
            _TRANSIT := TRUE;
            _STATE := STAMP_STATES_T#STAMP_INIT_4;
        END_IF;

    STAMP_STATES_T#STAMP_INIT_4:
        _TRANSIT := FALSE;
        STAMPPUSHER := FALSE;
        IF STAMPUP THEN
            _TRANSIT := TRUE;
            _STATE := STAMP_STATES_T#INTERSTEP;
        END_IF;

    STAMP_STATES_T#START_STAMP:
        _TRANSIT := FALSE;
        STAMPSLIDERMOVEDOUT := FALSE;
        STAMPSLIDERMOVEDIN := FALSE;
        STAMPPUSHER := FALSE;
        STAMPGREENLAMP := FALSE;
        STAMPPRESSURE := FALSE;
        STARTCOMMANDSTAMP := FALSE;
        IF (STAMPSTARTBUTTON = TRUE) THEN
            INTERCONNECTSTAMPSTARTCOMMAND := TRUE;
        END_IF;
        IF INTERCONNECTSTAMPSTARTCOMMAND THEN
            _TRANSIT := TRUE;
            _STATE := STAMP_STATES_T#GREEN_LAMP;
        END_IF;

    STAMP_STATES_T#STEP0:
        _TRANSIT := FALSE;
        IF CRANEUP THEN
            _TRANSIT := TRUE;
            _STATE := STAMP_STATES_T#STAMPSLIDERBACK;
        END_IF;

    STAMP_STATES_T#STEP1:
        _TRANSIT := FALSE;
        TIMER(IN := STAMPLOWERED, PT := TIME#12MS);
        INTERCONNECT := TIMER.Q;
        IF INTERCONNECT THEN
            _TRANSIT := TRUE;
            _STATE := STAMP_STATES_T#STAMPSLIDERFORWARD;
        END_IF;

    STAMP_STATES_T#STEP2:
        _TRANSIT := FALSE;
        IF (CRANEONCONVEYOR AND NOT STAMPSLIDERFILLED) THEN
            _TRANSIT := TRUE;
            _STATE := STAMP_STATES_T#INTERSTEP;
        END_IF;

    END_CASE;
END_FUNCTION_BLOCK

FUNCTION_BLOCK CRANE_FB
VAR  CRANTURNCLOCKWISE : BOOL; END_VAR
VAR_INPUT  CRANEDOWN : BOOL; END_VAR
VAR_OUTPUT  CRANELOWER : BOOL; END_VAR
VAR_INPUT  CRANEONCONVEYOR : BOOL; END_VAR
VAR_INPUT  CRANEONMAGAZIN : BOOL; END_VAR
VAR_INPUT  CRANEPOSITIONSTAMP : BOOL; END_VAR
VAR_INPUT  CRANESUCKED : BOOL; END_VAR
VAR_OUTPUT  CRANETURNCLOCKWISE : BOOL; END_VAR
VAR_OUTPUT  CRANETURNCOUNTERCLOCKWISE : BOOL; END_VAR
VAR_INPUT  CRANEUP : BOOL; END_VAR
VAR  DURATION1 : TIME := TIME#1S500MS; END_VAR
VAR_INPUT  MAGAZINCAPACITIVESENSOR : BOOL; END_VAR
VAR_OUTPUT  MAGAZINSLIDER : BOOL; END_VAR
VAR_OUTPUT  MAGAZINVACUUMOFF : BOOL; END_VAR
VAR_OUTPUT  MAGAZINVACUUMON : BOOL; END_VAR
VAR  SFCINIT : BOOL; END_VAR
VAR_INPUT  SFCRESET : BOOL; END_VAR
VAR_INPUT  SLIDERMOVEDOUT : BOOL; END_VAR
VAR_INPUT  SLIDERNOTMOVEDOUT : BOOL; END_VAR
VAR_INPUT  STAMPLOWERED : BOOL; END_VAR
VAR_INPUT  STAMPSLIDERFILLED : BOOL; END_VAR
VAR_INPUT  STARTBUTTONMAGAZIN : BOOL; END_VAR
VAR_OUTPUT  STARTCOMMANDCRANE : BOOL; END_VAR
VAR_INPUT  STARTVAR : BOOL; END_VAR
VAR  TIMEDELAY_TIMER : TON; END_VAR
VAR  TIMEDELAY_TIMER_DURATION : TIME := TIME#50MS; END_VAR
VAR  TIMEDELAY_TIMER_INTERCONNECT : BOOL; END_VAR
VAR  TIMER1 : TON; END_VAR
VAR_INPUT  WORKPIECEREADY : BOOL; END_VAR
VAR  _STATE : CRANE_STATES_T; END_VAR
VAR  _TRANSIT : BOOL; END_VAR
VAR  ACTUALTIME1 : TIME; END_VAR
VAR  INTERCONNECT : BOOL; END_VAR
VAR  INTERCONNECTCRANESTARTCOMMAND : BOOL; END_VAR

CASE _STATE OF
    CRANE_STATES_T#CRANE_GO_UP:
        _TRANSIT := FALSE;
        CRANELOWER := FALSE;
        IF (CRANEUP AND (MAGAZINCAPACITIVESENSOR OR NOT WORKPIECEREADY)) THEN
            _TRANSIT := TRUE;
            _STATE := CRANE_STATES_T#PAUSE;
        ELSIF ((CRANEUP AND NOT MAGAZINCAPACITIVESENSOR) AND WORKPIECEREADY) THEN
            _TRANSIT := TRUE;
            _STATE := CRANE_STATES_T#TURN_RIGHT_BLACK;
        END_IF;

    CRANE_STATES_T#CRANE_INIT:
        _TRANSIT := FALSE;
        CRANELOWER := TRUE;
        INTERCONNECTCRANESTARTCOMMAND := FALSE;
        IF CRANEDOWN THEN
            _TRANSIT := TRUE;
            _STATE := CRANE_STATES_T#CRANE_INIT_2;
        END_IF;

    CRANE_STATES_T#CRANE_INIT_2:
        _TRANSIT := FALSE;
        CRANELOWER := FALSE;
        IF CRANEUP THEN
            _TRANSIT := TRUE;
            _STATE := CRANE_STATES_T#INTERSTEP;
        END_IF;

    CRANE_STATES_T#CRANE_LIFT_AT_STAMP:
        _TRANSIT := FALSE;
        CRANELOWER := FALSE;
        IF CRANEUP THEN
            _TRANSIT := TRUE;
            _STATE := CRANE_STATES_T#CRANE_TURN_LEFT_FROM_STAMP;
        END_IF;

    CRANE_STATES_T#CRANE_LIFT_CONVEYOR:
        _TRANSIT := FALSE;
        CRANELOWER := FALSE;
        IF TRUE THEN
            _TRANSIT := TRUE;
            _STATE := CRANE_STATES_T#INTERSTEP;
        END_IF;

    CRANE_STATES_T#CRANE_LIFT_CONVEYOR_BLACK:
        _TRANSIT := FALSE;
        CRANELOWER := FALSE;
        IF CRANEUP THEN
            _TRANSIT := TRUE;
            _STATE := CRANE_STATES_T#CRANE_TURN_LEFT_BACK_TO_STAMP;
        END_IF;

    CRANE_STATES_T#CRANE_LIFT_MAGAZIN:
        _TRANSIT := FALSE;
        CRANELOWER := FALSE;
        IF CRANEUP THEN
            _TRANSIT := TRUE;
            _STATE := CRANE_STATES_T#CRANE_TURN_LEFT_NOT_METALLIC;
        END_IF;

    CRANE_STATES_T#CRANE_LIFT_MAGAZIN_METALLIC:
        _TRANSIT := FALSE;
        CRANELOWER := FALSE;
        IF CRANEUP THEN
            _TRANSIT := TRUE;
            _STATE := CRANE_STATES_T#CRANE_TURN_LEFT_METALLIC;
        END_IF;

    CRANE_STATES_T#CRANE_LIFT_NOT_METALLIC_BLACK:
        _TRANSIT := FALSE;
        CRANELOWER := FALSE;
        IF CRANEUP THEN
            _TRANSIT := TRUE;
            _STATE := CRANE_STATES_T#CRANE_TURN_LEFT_NOT_METALLIC_BLACK;
        END_IF;

    CRANE_STATES_T#CRANE_LOWER:
        _TRANSIT := FALSE;
        MAGAZINVACUUMON := TRUE;
        MAGAZINVACUUMOFF := FALSE;
        CRANELOWER := TRUE;
        IF CRANESUCKED THEN
            _TRANSIT := TRUE;
            _STATE := CRANE_STATES_T#STEP0;
        END_IF;

    CRANE_STATES_T#CRANE_ON_CONVEYOR:
        _TRANSIT := FALSE;
        CRANETURNCOUNTERCLOCKWISE := FALSE;
        CRANETURNCLOCKWISE := FALSE;
        CRANELOWER := TRUE;
        IF CRANEDOWN THEN
            _TRANSIT := TRUE;
            _STATE := CRANE_STATES_T#RELEASE;
        END_IF;

    CRANE_STATES_T#CRANE_ON_CONVEYOR_METALLIC:
        _TRANSIT := FALSE;
        CRANETURNCOUNTERCLOCKWISE := FALSE;
        CRANETURNCLOCKWISE := FALSE;
        CRANELOWER := TRUE;
        IF CRANEDOWN THEN
            _TRANSIT := TRUE;
            _STATE := CRANE_STATES_T#RELEASE;
        END_IF;

    CRANE_STATES_T#CRANE_ON_CONVEYOR_NOT_METALLICA_BLACK:
        _TRANSIT := FALSE;
        CRANETURNCOUNTERCLOCKWISE := FALSE;
        CRANETURNCLOCKWISE := FALSE;
        CRANELOWER := TRUE;
        IF CRANEDOWN THEN
            _TRANSIT := TRUE;
            _STATE := CRANE_STATES_T#RELEASE_BLACK;
        END_IF;

    CRANE_STATES_T#CRANE_ON_STAMP_METALLIC:
        _TRANSIT := FALSE;
        CRANETURNCOUNTERCLOCKWISE := FALSE;
        CRANETURNCLOCKWISE := FALSE;
        CRANELOWER := TRUE;
        IF CRANEDOWN THEN
            _TRANSIT := TRUE;
            _STATE := CRANE_STATES_T#RELEASE_WORKPIECE;
        END_IF;

    CRANE_STATES_T#CRANE_ON_STAMP_STOP_BLACK:
        _TRANSIT := FALSE;
        CRANETURNCLOCKWISE := FALSE;
        CRANETURNCOUNTERCLOCKWISE := FALSE;
        IF TRUE THEN
            _TRANSIT := TRUE;
            _STATE := CRANE_STATES_T#RESET_INTERCONNECT;
        END_IF;

    CRANE_STATES_T#CRANE_TURN_LEFT_BACK_TO_STAMP:
        _TRANSIT := FALSE;
        CRANETURNCOUNTERCLOCKWISE := TRUE;
        CRANETURNCLOCKWISE := FALSE;
        IF CRANEPOSITIONSTAMP THEN
            _TRANSIT := TRUE;
            _STATE := CRANE_STATES_T#CRANE_ON_STAMP_STOP_BLACK;
        END_IF;

    CRANE_STATES_T#CRANE_TURN_LEFT_FROM_STAMP:
        _TRANSIT := FALSE;
        CRANETURNCLOCKWISE := TRUE;
        CRANETURNCOUNTERCLOCKWISE := FALSE;
        IF CRANEONCONVEYOR THEN
            _TRANSIT := TRUE;
            _STATE := CRANE_STATES_T#CRANE_ON_CONVEYOR_METALLIC;
        END_IF;

    CRANE_STATES_T#CRANE_TURN_LEFT_METALLIC:
        _TRANSIT := FALSE;
        CRANETURNCOUNTERCLOCKWISE := TRUE;
        CRANETURNCLOCKWISE := FALSE;
        IF CRANEPOSITIONSTAMP THEN
            _TRANSIT := TRUE;
            _STATE := CRANE_STATES_T#CRANE_ON_STAMP_METALLIC;
        END_IF;

    CRANE_STATES_T#CRANE_TURN_LEFT_NOT_METALLIC:
        _TRANSIT := FALSE;
        CRANETURNCOUNTERCLOCKWISE := TRUE;
        CRANETURNCLOCKWISE := FALSE;
        IF CRANEONCONVEYOR THEN
            _TRANSIT := TRUE;
            _STATE := CRANE_STATES_T#CRANE_ON_CONVEYOR;
        END_IF;

    CRANE_STATES_T#CRANE_TURN_LEFT_NOT_METALLIC_BLACK:
        _TRANSIT := FALSE;
        CRANETURNCOUNTERCLOCKWISE := TRUE;
        CRANETURNCLOCKWISE := FALSE;
        IF CRANEONCONVEYOR THEN
            _TRANSIT := TRUE;
            _STATE := CRANE_STATES_T#CRANE_ON_CONVEYOR_NOT_METALLICA_BLACK;
        END_IF;

    CRANE_STATES_T#INIT:
        _TRANSIT := FALSE;
        IF TRUE THEN
            _TRANSIT := TRUE;
            _STATE := CRANE_STATES_T#START_CRANE;
        END_IF;

    CRANE_STATES_T#INTERSTEP:
        _TRANSIT := FALSE;
        STARTCOMMANDCRANE := TRUE;
        IF STARTVAR THEN
            _TRANSIT := TRUE;
            _STATE := CRANE_STATES_T#INTERSTEP_2;
        END_IF;

    CRANE_STATES_T#INTERSTEP_2:
        _TRANSIT := FALSE;
        IF SLIDERMOVEDOUT THEN
            _TRANSIT := TRUE;
            _STATE := CRANE_STATES_T#TIMEDELAY;
        END_IF;

    CRANE_STATES_T#LAST_WORKPIECE_AT_STAMP:
        _TRANSIT := FALSE;
        IF TRUE THEN
            _TRANSIT := TRUE;
            _STATE := CRANE_STATES_T#PAUSE;
        END_IF;

    CRANE_STATES_T#LOWER_CRANE:
        _TRANSIT := FALSE;
        CRANELOWER := TRUE;
        IF CRANEDOWN THEN
            _TRANSIT := TRUE;
            _STATE := CRANE_STATES_T#SUCK_AT_STAMP;
        END_IF;

    CRANE_STATES_T#MAGAZIN_STOP:
        _TRANSIT := FALSE;
        CRANETURNCLOCKWISE := FALSE;
        CRANETURNCOUNTERCLOCKWISE := FALSE;
        IF (NOT WORKPIECEREADY AND NOT STAMPSLIDERFILLED) THEN
            _TRANSIT := TRUE;
            _STATE := CRANE_STATES_T#NO_WORKPIECE_READY;
        ELSIF WORKPIECEREADY THEN
            _TRANSIT := TRUE;
            _STATE := CRANE_STATES_T#CRANE_LOWER;
        ELSIF (NOT WORKPIECEREADY AND STAMPSLIDERFILLED) THEN
            _TRANSIT := TRUE;
            _STATE := CRANE_STATES_T#LAST_WORKPIECE_AT_STAMP;
        END_IF;

    CRANE_STATES_T#MAGAZIN_STOP_BLACK:
        _TRANSIT := FALSE;
        CRANETURNCLOCKWISE := FALSE;
        CRANETURNCOUNTERCLOCKWISE := FALSE;
        MAGAZINVACUUMON := TRUE;
        MAGAZINVACUUMOFF := FALSE;
        CRANELOWER := TRUE;
        IF CRANESUCKED THEN
            _TRANSIT := TRUE;
            _STATE := CRANE_STATES_T#CRANE_LIFT_NOT_METALLIC_BLACK;
        END_IF;

    CRANE_STATES_T#NO_WORKPIECE_READY:
        _TRANSIT := FALSE;
        IF TRUE THEN
            _TRANSIT := TRUE;
            _STATE := CRANE_STATES_T#START_CRANE;
        END_IF;

    CRANE_STATES_T#RESET_INTERCONNECT:
        _TRANSIT := FALSE;
        INTERCONNECT := FALSE;
        TIMER1(IN := FALSE, PT := TIME#1MS);
        IF SLIDERMOVEDOUT THEN
            _TRANSIT := TRUE;
            _STATE := CRANE_STATES_T#LOWER_CRANE;
        END_IF;

    CRANE_STATES_T#START_CRANE:
        _TRANSIT := FALSE;
        CRANELOWER := FALSE;
        MAGAZINVACUUMOFF := TRUE;
        MAGAZINVACUUMON := FALSE;
        CRANETURNCOUNTERCLOCKWISE := FALSE;
        CRANETURNCLOCKWISE := FALSE;
        STARTVAR := FALSE;
        STARTCOMMANDCRANE := FALSE;
        IF (STARTBUTTONMAGAZIN = TRUE) THEN
            INTERCONNECTCRANESTARTCOMMAND := TRUE;
        END_IF;
        IF INTERCONNECTCRANESTARTCOMMAND THEN
            _TRANSIT := TRUE;
            _STATE := CRANE_STATES_T#CRANE_INIT;
        END_IF;

    CRANE_STATES_T#STEP0:
        _TRANSIT := FALSE;
        IF NOT MAGAZINCAPACITIVESENSOR THEN
            _TRANSIT := TRUE;
            _STATE := CRANE_STATES_T#CRANE_LIFT_MAGAZIN;
        ELSIF MAGAZINCAPACITIVESENSOR THEN
            _TRANSIT := TRUE;
            _STATE := CRANE_STATES_T#CRANE_LIFT_MAGAZIN_METALLIC;
        END_IF;

    CRANE_STATES_T#SUCK_AT_STAMP:
        _TRANSIT := FALSE;
        MAGAZINVACUUMON := TRUE;
        MAGAZINVACUUMOFF := FALSE;
        IF CRANESUCKED THEN
            _TRANSIT := TRUE;
            _STATE := CRANE_STATES_T#CRANE_LIFT_AT_STAMP;
        END_IF;

    CRANE_STATES_T#TIMEDELAY:
        _TRANSIT := FALSE;
        TIMEDELAY_TIMER(IN := TRUE, PT := TIMEDELAY_TIMER_DURATION);
        TIMEDELAY_TIMER_INTERCONNECT := TIMEDELAY_TIMER.Q;
        IF TIMEDELAY_TIMER_INTERCONNECT THEN
            _TRANSIT := TRUE;
            _STATE := CRANE_STATES_T#TURN_RIGHT;
        END_IF;

    CRANE_STATES_T#TURN_RIGHT:
        _TRANSIT := FALSE;
        CRANETURNCLOCKWISE := TRUE;
        CRANETURNCOUNTERCLOCKWISE := FALSE;
        IF CRANEONMAGAZIN THEN
            _TRANSIT := TRUE;
            _STATE := CRANE_STATES_T#MAGAZIN_STOP;
        END_IF;

    CRANE_STATES_T#TURN_RIGHT_BLACK:
        _TRANSIT := FALSE;
        CRANETURNCLOCKWISE := TRUE;
        CRANETURNCOUNTERCLOCKWISE := FALSE;
        IF CRANEONMAGAZIN THEN
            _TRANSIT := TRUE;
            _STATE := CRANE_STATES_T#MAGAZIN_STOP_BLACK;
        END_IF;

    CRANE_STATES_T#PAUSE:
        _TRANSIT := FALSE;
        TIMER1(IN := CRANEUP, PT := DURATION1);
        INTERCONNECT := TIMER1.Q;
        IF INTERCONNECT THEN
            _TRANSIT := TRUE;
            _STATE := CRANE_STATES_T#RESET_INTERCONNECT;
        END_IF;

    CRANE_STATES_T#RELEASE:
        _TRANSIT := FALSE;
        MAGAZINVACUUMOFF := TRUE;
        MAGAZINVACUUMON := FALSE;
        IF TRUE THEN
            _TRANSIT := TRUE;
            _STATE := CRANE_STATES_T#CRANE_LIFT_CONVEYOR;
        END_IF;

    CRANE_STATES_T#RELEASE_BLACK:
        _TRANSIT := FALSE;
        MAGAZINVACUUMON := FALSE;
        MAGAZINVACUUMOFF := TRUE;
        IF TRUE THEN
            _TRANSIT := TRUE;
            _STATE := CRANE_STATES_T#CRANE_LIFT_CONVEYOR_BLACK;
        END_IF;

    CRANE_STATES_T#RELEASE_WORKPIECE:
        _TRANSIT := FALSE;
        MAGAZINVACUUMOFF := TRUE;
        MAGAZINVACUUMON := FALSE;
        IF TRUE THEN
            _TRANSIT := TRUE;
            _STATE := CRANE_STATES_T#CRANE_GO_UP;
        END_IF;

    END_CASE;
END_FUNCTION_BLOCK

PROGRAM MAIN

VAR_OUTPUT ACTUATOR_ANALOGCRANEPRESSURE : INT; END_VAR
VAR_OUTPUT ACTUATOR_CRANELOWER : BOOL; END_VAR
VAR_OUTPUT ACTUATOR_CRANETURNCLOCKWISE : BOOL; END_VAR
VAR_OUTPUT ACTUATOR_CRANETURNCOUNTERCLOCKWISE : BOOL; END_VAR
VAR_OUTPUT ACTUATOR_MAGAZINGREENLAMP : BOOL; END_VAR
VAR_OUTPUT ACTUATOR_MAGAZINSLIDER : BOOL; END_VAR
VAR_OUTPUT ACTUATOR_MAGAZINVACUUMOFF : BOOL; END_VAR
VAR_OUTPUT ACTUATOR_MAGAZINVACUUMON : BOOL; END_VAR
VAR_OUTPUT ACTUATOR_MAGAZINWHITELAMP : BOOL; END_VAR
VAR_OUTPUT ACTUATOR_STAMPGREENLAMP : BOOL; END_VAR
VAR_OUTPUT ACTUATOR_STAMPPUSHER : BOOL; END_VAR
VAR_OUTPUT ACTUATOR_STAMPSLIDERMOVEDIN : BOOL; END_VAR
VAR_OUTPUT ACTUATOR_STAMPSLIDERMOVEDOUT : BOOL; END_VAR
VAR_OUTPUT ACTUATOR_STAMPWHITELAMP : BOOL; END_VAR
VAR  CRANE : CRANE_FB; END_VAR
VAR  MAG : MAGAZIN; END_VAR
VAR_INPUT SENSOR_CRANEDOWN : BOOL; END_VAR
VAR_INPUT SENSOR_CRANEONCONVEYOR : BOOL; END_VAR
VAR_INPUT SENSOR_CRANEONMAGAZIN : BOOL; END_VAR
VAR_INPUT SENSOR_CRANEPOSITION : BOOL; END_VAR
VAR_INPUT SENSOR_CRANEPOSITIONSTAMP : BOOL; END_VAR
VAR_INPUT SENSOR_CRANESUCKED : BOOL; END_VAR
VAR_INPUT SENSOR_CRANEUP : BOOL; END_VAR
VAR_INPUT SENSOR_MAGAZINCAPACITIVESENSOR : BOOL; END_VAR
VAR_INPUT SENSOR_MAGAZINEMERGENCYSTOP : BOOL; END_VAR
VAR_INPUT SENSOR_MAGAZINOPTICALSENSOR : BOOL; END_VAR
VAR_INPUT SENSOR_MAGAZINSWITCHMANUELLAUTOMATIC : BOOL; END_VAR
VAR_INPUT SENSOR_SLIDERMOVEDOUT : BOOL; END_VAR
VAR_INPUT SENSOR_SLIDERNOTMOVEDOUT : BOOL; END_VAR
VAR_INPUT SENSOR_STAMPEMERGENCYSTOP : BOOL; END_VAR
VAR_INPUT SENSOR_STAMPLOWERED : BOOL; END_VAR
VAR_INPUT SENSOR_STAMPSLIDERFILLED : BOOL; END_VAR
VAR_INPUT SENSOR_STAMPSLIDERSENSORMOVEDIN : BOOL; END_VAR
VAR_INPUT SENSOR_STAMPSLIDERSENSORMOVEDOUT : BOOL; END_VAR
VAR_INPUT SENSOR_STAMPSTARTBUTTON : BOOL; END_VAR
VAR_INPUT SENSOR_STAMPSWITCHMANUELLAUTOMATIC : BOOL; END_VAR
VAR_INPUT SENSOR_STAMPUP : BOOL; END_VAR
VAR_INPUT SENSOR_STARTBUTTONMAGAZIN : BOOL; END_VAR
VAR_INPUT SENSOR_WORKPIECEREADY : BOOL; END_VAR
VAR  STAMP : STAMP_FB; END_VAR

CRANE.CRANEDOWN := SENSOR_CRANEDOWN;
CRANE.CRANEONCONVEYOR := SENSOR_CRANEONCONVEYOR;
CRANE.CRANEONMAGAZIN := SENSOR_CRANEONMAGAZIN;
CRANE.CRANEPOSITIONSTAMP := SENSOR_CRANEPOSITIONSTAMP;
CRANE.CRANESUCKED := SENSOR_CRANESUCKED;
CRANE.CRANEUP := SENSOR_CRANEUP;
CRANE.MAGAZINCAPACITIVESENSOR := SENSOR_MAGAZINCAPACITIVESENSOR;
CRANE.SLIDERMOVEDOUT := SENSOR_SLIDERMOVEDOUT;
CRANE.STAMPSLIDERFILLED := SENSOR_STAMPSLIDERFILLED;
CRANE.STARTBUTTONMAGAZIN := SENSOR_STARTBUTTONMAGAZIN;
CRANE.WORKPIECEREADY := SENSOR_WORKPIECEREADY;
MAG.CRANEDOWN := SENSOR_CRANEDOWN;
MAG.CRANEONCONVEYOR := SENSOR_CRANEONCONVEYOR;
MAG.CRANEONMAGAZIN := SENSOR_CRANEONMAGAZIN;
MAG.CRANEUP := SENSOR_CRANEUP;
MAG.SLIDERMOVEDOUT := SENSOR_SLIDERMOVEDOUT;
MAG.SLIDERNOTMOVEDOUT := SENSOR_SLIDERNOTMOVEDOUT;
MAG.STARTBUTTONMAGAZIN := SENSOR_STARTBUTTONMAGAZIN;
MAG.WORKPIECEREADY := SENSOR_WORKPIECEREADY;
STAMP.CRANEDOWN := SENSOR_CRANEDOWN;
STAMP.CRANEONCONVEYOR := SENSOR_CRANEONCONVEYOR;
STAMP.CRANEPOSITIONSTAMP := SENSOR_CRANEPOSITIONSTAMP;
STAMP.CRANESUCKED := SENSOR_CRANESUCKED;
STAMP.CRANEUP := SENSOR_CRANEUP;
STAMP.STAMPLOWERED := SENSOR_STAMPLOWERED;
STAMP.STAMPSLIDERFILLED := SENSOR_STAMPSLIDERFILLED;
STAMP.STAMPSLIDERSENSORMOVEDIN := SENSOR_STAMPSLIDERSENSORMOVEDIN;
STAMP.STAMPSLIDERSENSORMOVEDOUT := SENSOR_STAMPSLIDERSENSORMOVEDOUT;
STAMP.STAMPSTARTBUTTON := SENSOR_STAMPSTARTBUTTON;
STAMP.STAMPUP := SENSOR_STAMPUP;

IF (SENSOR_STAMPEMERGENCYSTOP AND SENSOR_MAGAZINEMERGENCYSTOP) THEN
    MAG();
    CRANE();
    STAMP();
    IF (ACTUATOR_MAGAZINGREENLAMP AND ACTUATOR_STAMPGREENLAMP) THEN
        IF ((STAMP.STARTCOMMANDSTAMP AND CRANE.STARTCOMMANDCRANE) AND MAG.STARTCOMMANDMAGAZIN) THEN
            CRANE.STARTVAR := TRUE;
            MAG.STARTVAR := TRUE;
            STAMP.STARTVAR := TRUE;
        END_IF;
    END_IF;
    CRANE.SFCRESET := FALSE;
    MAG.SFCRESET := FALSE;
    STAMP.SFCRESET := FALSE;

    ACTUATOR_ANALOGCRANEPRESSURE := INT#6000;
    ACTUATOR_CRANELOWER := CRANE.CRANELOWER;
    ACTUATOR_CRANETURNCLOCKWISE := CRANE.CRANETURNCLOCKWISE;
    ACTUATOR_CRANETURNCOUNTERCLOCKWISE := CRANE.CRANETURNCOUNTERCLOCKWISE;
    ACTUATOR_MAGAZINGREENLAMP := MAG.MAGAZINGREENLAMP;
    ACTUATOR_MAGAZINSLIDER := MAG.MAGAZINSLIDER;
    ACTUATOR_MAGAZINVACUUMOFF := CRANE.MAGAZINVACUUMOFF;
    ACTUATOR_MAGAZINVACUUMON := CRANE.MAGAZINVACUUMON;
    ACTUATOR_STAMPGREENLAMP := STAMP.STAMPGREENLAMP;
    ACTUATOR_STAMPPUSHER := STAMP.STAMPPUSHER;
    ACTUATOR_STAMPSLIDERMOVEDIN := STAMP.STAMPSLIDERMOVEDIN;
    ACTUATOR_STAMPSLIDERMOVEDOUT := STAMP.STAMPSLIDERMOVEDOUT;
    ACTUATOR_STAMPWHITELAMP := STAMP.STAMPWHITELAMP;

ELSIF (NOT SENSOR_STAMPEMERGENCYSTOP OR NOT SENSOR_MAGAZINEMERGENCYSTOP) THEN
    ACTUATOR_MAGAZINSLIDER := FALSE;
    ACTUATOR_CRANELOWER := FALSE;
    ACTUATOR_MAGAZINVACUUMON := FALSE;
    ACTUATOR_MAGAZINVACUUMOFF := TRUE;
    ACTUATOR_MAGAZINGREENLAMP := FALSE;
    ACTUATOR_CRANETURNCOUNTERCLOCKWISE := FALSE;
    ACTUATOR_CRANETURNCLOCKWISE := FALSE;
    ACTUATOR_STAMPSLIDERMOVEDOUT := TRUE;
    ACTUATOR_STAMPSLIDERMOVEDIN := FALSE;
    ACTUATOR_STAMPGREENLAMP := FALSE;
    ACTUATOR_STAMPPUSHER := FALSE;
    ACTUATOR_ANALOGCRANEPRESSURE := INT#0;
    CRANE.SFCRESET := TRUE;
    MAG.SFCRESET := TRUE;
    STAMP.SFCRESET := TRUE;
    CRANE.STARTVAR := FALSE;
    MAG.STARTVAR := FALSE;
    STAMP.STARTVAR := FALSE;
END_IF;
END_PROGRAM

CONFIGURATION Config0
  RESOURCE Res0 ON PLC
    TASK TASK0(INTERVAL := T#50MS, PRIORITY := 0);
    PROGRAM INSTANCE0 WITH TASK0 : MAIN;
  END_RESOURCE
END_CONFIGURATION

(* ---- program.st ---- *)
FUNCTION_BLOCK FB
VAR_INPUT
	x : INT;
END_VAR
VAR_OUTPUT
	y : INT;
END_VAR
	y := x+6;
END_FUNCTION_BLOCK

PROGRAM PGRM
VAR_INPUT
	x : INT;
END_VAR
VAR_OUTPUT
	y : INT;
END_VAR
VAR
	INST_FB : FB;
END_VAR
	INST_FB.x := 4;
	INST_FB();
	INST_FB.x := INST_FB.y + 2;
	INST_FB();
	y := INST_FB.y;
	IF x > 5 THEN
		y := 6;
	ELSIF x > 3 THEN
		y := 7;
	ELSE
		y := x;
	END_IF;
	y := y + 4;
END_PROGRAM
CONFIGURATION Config0
  RESOURCE Res0 ON PLC
    TASK task0(INTERVAL := T#50ms, PRIORITY := 0);
    PROGRAM instance0 WITH task0 : PGRM;
  END_RESOURCE
END_CONFIGURATION

(* ---- program1_wMan.st ---- *)
TYPE
	TESTENUM: (FIRST, SECOND);
END_TYPE

FUNCTION_BLOCK BLOCK_A
	VAR_INPUT  X : INT; END_VAR
	VAR_OUTPUT Y : INT; END_VAR
	Y := X - INT#4;
END_FUNCTION_BLOCK

FUNCTION_BLOCK BLOCK_B
	VAR_INPUT  X : INT; END_VAR
	VAR_OUTPUT Y : INT; END_VAR
	Y := X + INT#6;
END_FUNCTION_BLOCK

PROGRAM PGRM
	VAR_INPUT  X      : INT;     END_VAR
	VAR_OUTPUT Y      : INT;     END_VAR
	VAR        INST_A : BLOCK_A; END_VAR
	VAR        INST_B : BLOCK_B; END_VAR
	VAR        STATE  : TESTENUM; END_VAR
	VAR  TESTTIMER : TON; END_VAR

	CASE STATE OF
		TESTENUM#FIRST:
			INST_A.X := INT#4;
		TESTENUM#SECOND:
			INST_A.X := INT#8;
	END_CASE;
	TESTTIMER();
	INST_A.X := X + INT#7;
	IF X > 5 THEN
		INST_A();
	END_IF;

	INST_B.X := INST_A.Y + INT#9;
	INST_B();

	Y := INST_B.Y;
END_PROGRAM

CONFIGURATION Config0
  RESOURCE Res0 ON PLC
    TASK TASK0(INTERVAL := T#50MS, PRIORITY := 0);
    PROGRAM INSTANCE0 WITH TASK0 : PGRM;
  END_RESOURCE
END_CONFIGURATION

(* ---- program2.st ---- *)
FUNCTION_BLOCK BLOCK_A
	VAR_INPUT  X : INT; END_VAR
	VAR_OUTPUT Y : INT; END_VAR
	Y := X - INT#4;
END_FUNCTION_BLOCK

FUNCTION_BLOCK BLOCK_B
	VAR_INPUT  X : INT; END_VAR
	VAR_OUTPUT Y : INT; END_VAR
	Y := X + INT#3;
END_FUNCTION_BLOCK

PROGRAM PGRM
	VAR_INPUT  X      : INT;     END_VAR
	VAR_OUTPUT Y      : INT;     END_VAR
	VAR        INST_A : BLOCK_A; END_VAR
	VAR        INST_B : BLOCK_B; END_VAR

	INST_A.X := X + INT#7;
	INST_A();

	INST_B.X := INST_A.Y + INT#9;
	INST_B();

	Y := INST_B.Y + INT#3;
END_PROGRAM

CONFIGURATION Config0
  RESOURCE Res0 ON PLC
    TASK TASK0(INTERVAL := T#50MS, PRIORITY := 0);
    PROGRAM INSTANCE0 WITH TASK0 : PGRM;
  END_RESOURCE
END_CONFIGURATION

(* ---- runtimeTest.functionBlockTest.st ---- *)
FUNCTION_BLOCK TON_B

VAR_INPUT
    IN : BOOL;
    IN2 : BOOL;
END_VAR

VAR_OUTPUT
    Q  : BOOL := TRUE;
END_VAR

    Q := IN AND IN2;

END_FUNCTION_BLOCK

PROGRAM  Analogsensor

    VAR
      timeout          	: TON_B;
      e : BOOL;
    END_VAR

    timeout(IN := TRUE, IN2 := TRUE);

    e := timeout.Q;

END_PROGRAM

CONFIGURATION Config0
  RESOURCE Res0 ON PLC
    TASK task0(INTERVAL := T#50ms, PRIORITY := 0);
    PROGRAM instance0 WITH task0 : Analogsensor;
  END_RESOURCE
END_CONFIGURATION

(* ---- scenario0.st ---- *)
TYPE
    Magazin_states_t : (Green_Lamp , Init , Interstep , Magazin_Init , Magazin_Init_2 , Slider_Move_Back , Start_Magazin , Step0 , Step1 , convey);
    Crane_states_t : (Crane_Init , Crane_Init_2 , Crane_Lift_Conveyor , Crane_Lift_Magazine , Crane_On_Conveyor , Crane_Stop , Crane_Turn_Left , Init , Interstep , Interstep_2 , Interstep_Check_Workpiece , Magazin_Stop , Start_Crane , TimeDelay , Turn_Right , release);
END_TYPE

FUNCTION_BLOCK Magazin
    VAR_INPUT  CraneDown : BOOL; END_VAR
    VAR_INPUT  CraneOnConveyor : BOOL; END_VAR
    VAR_INPUT  CraneOnMagazin : BOOL; END_VAR
    VAR_INPUT  CraneSucked : BOOL; END_VAR
    VAR_INPUT  CraneUp : BOOL; END_VAR
    VAR_OUTPUT  MagazinGreenLamp : BOOL; END_VAR
    VAR_OUTPUT  MagazinSlider : BOOL; END_VAR
    VAR  SFCInit : BOOL; END_VAR
    VAR_INPUT  SFCReset : BOOL; END_VAR
    VAR_INPUT  SliderMovedOut : BOOL; END_VAR
    VAR_INPUT  SliderNotMovedOut : BOOL; END_VAR
    VAR_INPUT  StartButtonMagazin : BOOL; END_VAR
    VAR_OUTPUT  StartCommandMagazin : BOOL; END_VAR
    VAR_INPUT  StartVar : BOOL; END_VAR
    VAR_INPUT  WorkpieceReady : BOOL; END_VAR
    VAR  _state : Magazin_states_t; END_VAR
    VAR  _transit : BOOL; END_VAR
    VAR  interconnectMagazineStartCommand : BOOL; END_VAR

    CASE _state OF
        Magazin_states_t#Green_Lamp:
            _transit := FALSE;
            MagazinGreenLamp := TRUE;
            interconnectMagazineStartCommand := FALSE;
            IF TRUE THEN
                _transit := TRUE;
                _state := Magazin_states_t#Magazin_Init;
            END_IF;

        Magazin_states_t#Init:
            _transit := FALSE;
            IF TRUE THEN
                _transit := TRUE;
                _state := Magazin_states_t#Start_Magazin;
            END_IF;

        Magazin_states_t#Interstep:
            _transit := FALSE;
            StartCommandMagazin := TRUE;
            IF StartVar THEN
                _transit := TRUE;
                _state := Magazin_states_t#convey;
            END_IF;

        Magazin_states_t#Magazin_Init:
            _transit := FALSE;
            MagazinSlider := TRUE;
            IF TRUE THEN
                _transit := TRUE;
                _state := Magazin_states_t#Magazin_Init_2;
            END_IF;

        Magazin_states_t#Magazin_Init_2:
            _transit := FALSE;
            MagazinSlider := FALSE;
            IF TRUE THEN
                _transit := TRUE;
                _state := Magazin_states_t#Interstep;
            END_IF;

        Magazin_states_t#Slider_Move_Back:
            _transit := FALSE;
            IF ((SliderMovedOut = TRUE) AND (SliderNotMovedOut = FALSE)) THEN
                MagazinSlider := FALSE;
            END_IF;
            IF CraneUp THEN
                _transit := TRUE;
                _state := Magazin_states_t#Step1;
            END_IF;

        Magazin_states_t#Start_Magazin:
            _transit := FALSE;
            MagazinSlider := FALSE;
            MagazinGreenLamp := FALSE;
            StartVar := FALSE;
            StartCommandMagazin := FALSE;
            IF (StartButtonMagazin = TRUE) THEN
                interconnectMagazineStartCommand := TRUE;
            END_IF;
            IF interconnectMagazineStartCommand THEN
                _transit := TRUE;
                _state := Magazin_states_t#Green_Lamp;
            END_IF;

        Magazin_states_t#Step0:
            _transit := FALSE;
            IF CraneDown THEN
                _transit := TRUE;
                _state := Magazin_states_t#Slider_Move_Back;
            END_IF;

        Magazin_states_t#Step1:
            _transit := FALSE;
            IF CraneOnConveyor THEN
                _transit := TRUE;
                _state := Magazin_states_t#Interstep;
            END_IF;

        Magazin_states_t#convey:
            _transit := FALSE;
            IF SliderNotMovedOut THEN
                MagazinSlider := TRUE;
            END_IF;
            IF CraneOnMagazin THEN
                _transit := TRUE;
                _state := Magazin_states_t#Step0;
            END_IF;

            END_CASE;
END_FUNCTION_BLOCK

FUNCTION_BLOCK Crane_FB
    VAR_INPUT  CraneDown : BOOL; END_VAR
    VAR_OUTPUT  CraneLower : BOOL; END_VAR
    VAR_INPUT  CraneOnConveyor : BOOL; END_VAR
    VAR_INPUT  CraneOnMagazin : BOOL; END_VAR
    VAR_INPUT  CraneSucked : BOOL; END_VAR
    VAR_OUTPUT  CraneTurnClockwise : BOOL; END_VAR
    VAR_OUTPUT  CraneTurnCounterclockwise : BOOL; END_VAR
    VAR_INPUT  CraneUp : BOOL; END_VAR
    VAR_OUTPUT  MagazinVacuumOff : BOOL; END_VAR
    VAR_OUTPUT  MagazinVacuumOn : BOOL; END_VAR
    VAR  SFCInit : BOOL; END_VAR
    VAR_INPUT  SFCReset : BOOL; END_VAR
    VAR_INPUT  SliderMovedOut : BOOL; END_VAR
    VAR_INPUT  SliderNotMovedOut : BOOL; END_VAR
    VAR_INPUT  StartButtonMagazin : BOOL; END_VAR
    VAR_OUTPUT  StartCommandCrane : BOOL; END_VAR
    VAR_INPUT  StartVar : BOOL; END_VAR
    VAR  TimeDelay_Timer : TON; END_VAR
    VAR  TimeDelay_Timer_Duration : INT := INT#50; END_VAR
    VAR  TimeDelay_Timer_interconnect : BOOL; END_VAR
    VAR_INPUT  WorkpieceReady : BOOL; END_VAR
    VAR  _state : Crane_states_t; END_VAR
    VAR  _transit : BOOL; END_VAR
    VAR  interconnectCraneStartCommand : BOOL; END_VAR

    CASE _state OF
        Crane_states_t#Crane_Init:
            _transit := FALSE;
            CraneLower := TRUE;
            interconnectCraneStartCommand := FALSE;
            IF CraneDown THEN
                _transit := TRUE;
                _state := Crane_states_t#Crane_Init_2;
            END_IF;

        Crane_states_t#Crane_Init_2:
            _transit := FALSE;
            CraneLower := FALSE;
            IF CraneUp THEN
                _transit := TRUE;
                _state := Crane_states_t#Interstep;
            END_IF;

        Crane_states_t#Crane_Lift_Conveyor:
            _transit := FALSE;
            CraneLower := FALSE;
            IF TRUE THEN
                _transit := TRUE;
                _state := Crane_states_t#Interstep;
            END_IF;

        Crane_states_t#Crane_Lift_Magazine:
            _transit := FALSE;
            CraneLower := FALSE;
            IF CraneUp THEN
                _transit := TRUE;
                _state := Crane_states_t#Crane_Turn_Left;
            END_IF;

        Crane_states_t#Crane_On_Conveyor:
            _transit := FALSE;
            CraneTurnCounterclockwise := FALSE;
            CraneTurnClockwise := FALSE;
            CraneLower := TRUE;
            IF CraneDown THEN
                _transit := TRUE;
                _state := Crane_states_t#release;
            END_IF;

        Crane_states_t#Crane_Stop:
            _transit := FALSE;
            IF TRUE THEN
                _transit := TRUE;
                _state := Crane_states_t#Start_Crane;
            END_IF;

        Crane_states_t#Crane_Turn_Left:
            _transit := FALSE;
            CraneTurnCounterclockwise := TRUE;
            CraneTurnClockwise := FALSE;
            IF CraneOnConveyor THEN
                _transit := TRUE;
                _state := Crane_states_t#Crane_On_Conveyor;
            END_IF;

        Crane_states_t#Init:
            _transit := FALSE;
            IF TRUE THEN
                _transit := TRUE;
                _state := Crane_states_t#Start_Crane;
            END_IF;

        Crane_states_t#Interstep:
            _transit := FALSE;
            StartCommandCrane := TRUE;
            IF StartVar THEN
                _transit := TRUE;
                _state := Crane_states_t#Interstep_2;
            END_IF;

        Crane_states_t#Interstep_2:
            _transit := FALSE;
            IF SliderMovedOut THEN
                _transit := TRUE;
                _state := Crane_states_t#TimeDelay;
            END_IF;

        Crane_states_t#Interstep_Check_Workpiece:
            _transit := FALSE;
            IF WorkpieceReady THEN
                _transit := TRUE;
                _state := Crane_states_t#Magazin_Stop;
            ELSIF NOT WorkpieceReady THEN
                _transit := TRUE;
                _state := Crane_states_t#Crane_Stop;
            END_IF;

        Crane_states_t#Magazin_Stop:
            _transit := FALSE;
            CraneTurnClockwise := FALSE;
            CraneTurnCounterclockwise := FALSE;
            MagazinVacuumOn := TRUE;
            MagazinVacuumOff := FALSE;
            CraneLower := TRUE;
            IF CraneSucked THEN
                _transit := TRUE;
                _state := Crane_states_t#Crane_Lift_Magazine;
            END_IF;

        Crane_states_t#Start_Crane:
            _transit := FALSE;
            CraneLower := FALSE;
            MagazinVacuumOff := TRUE;
            MagazinVacuumOn := FALSE;
            CraneTurnCounterclockwise := FALSE;
            CraneTurnClockwise := FALSE;
            StartVar := FALSE;
            StartCommandCrane := FALSE;
            IF (StartButtonMagazin = TRUE) THEN
                interconnectCraneStartCommand := TRUE;
            END_IF;
            IF interconnectCraneStartCommand THEN
                _transit := TRUE;
                _state := Crane_states_t#Crane_Init;
            END_IF;

        Crane_states_t#TimeDelay:
            _transit := FALSE;
            TimeDelay_Timer(IN := TRUE, PT := INT_TO_TIME(TimeDelay_Timer_Duration));
            TimeDelay_Timer_interconnect := TimeDelay_Timer.Q;
            IF TimeDelay_Timer_interconnect THEN
                _transit := TRUE;
                _state := Crane_states_t#Turn_Right;
            END_IF;

        Crane_states_t#Turn_Right:
            _transit := FALSE;
            CraneTurnClockwise := TRUE;
            CraneTurnCounterclockwise := FALSE;
            IF CraneOnMagazin THEN
                _transit := TRUE;
                _state := Crane_states_t#Interstep_Check_Workpiece;
            END_IF;

        Crane_states_t#release:
            _transit := FALSE;
            MagazinVacuumOff := TRUE;
            MagazinVacuumOn := FALSE;
            IF TRUE THEN
                _transit := TRUE;
                _state := Crane_states_t#Crane_Lift_Conveyor;
            END_IF;

            END_CASE;
END_FUNCTION_BLOCK

PROGRAM Main

VAR_OUTPUT  Actuator_CraneLower : BOOL; END_VAR
VAR_OUTPUT  Actuator_CraneTurnClockwise : BOOL; END_VAR
VAR_OUTPUT  Actuator_CraneTurnCounterclockwise : BOOL; END_VAR
VAR_OUTPUT  Actuator_MagazinGreenLamp : BOOL; END_VAR
VAR_OUTPUT  Actuator_MagazinSlider : BOOL; END_VAR
VAR_OUTPUT  Actuator_MagazinVacuumOff : BOOL; END_VAR
VAR_OUTPUT  Actuator_MagazinVacuumOn : BOOL; END_VAR
VAR_OUTPUT  Actuator_MagazinWhiteLamp : BOOL; END_VAR
VAR  Crane : Crane_FB; END_VAR
VAR  Mag : Magazin; END_VAR
VAR_INPUT  Sensor_CraneDown : BOOL; END_VAR
VAR_INPUT  Sensor_CraneOnConveyor : BOOL; END_VAR
VAR_INPUT  Sensor_CraneOnMagazin : BOOL; END_VAR
VAR_INPUT  Sensor_CranePosition : BOOL; END_VAR
VAR_INPUT  Sensor_CraneSucked : BOOL; END_VAR
VAR_INPUT  Sensor_CraneUp : BOOL; END_VAR
VAR_INPUT  Sensor_MagazinEmergencyStop : BOOL; END_VAR
VAR_INPUT  Sensor_MagazinSwitchManuellAutomatic : BOOL; END_VAR
VAR_INPUT  Sensor_SliderMovedOut : BOOL; END_VAR
VAR_INPUT  Sensor_SliderNotMovedOut : BOOL; END_VAR
VAR_INPUT  Sensor_StartButtonMagazin : BOOL; END_VAR
VAR_INPUT  Sensor_WorkpieceReady : BOOL; END_VAR
Mag.SliderNotMovedOut := Sensor_SliderNotMovedOut;
Mag.SliderMovedOut := Sensor_SliderMovedOut;
Mag.CraneOnMagazin := Sensor_CraneOnMagazin;
Mag.CraneDown := Sensor_CraneDown;
Mag.CraneUp := Sensor_CraneUp;
Mag.CraneOnConveyor := Sensor_CraneOnConveyor;
Mag.WorkpieceReady := Sensor_WorkpieceReady;
Mag.StartButtonMagazin := Sensor_StartButtonMagazin;
Actuator_MagazinSlider := Mag.MagazinSlider;
Actuator_MagazinGreenLamp := Mag.MagazinGreenLamp;
Crane.WorkpieceReady := Sensor_WorkpieceReady;
Crane.CraneUp := Sensor_CraneUp;
Crane.CraneOnConveyor := Sensor_CraneOnConveyor;
Crane.CraneDown := Sensor_CraneDown;
Crane.CraneSucked := Sensor_CraneSucked;
Crane.CraneOnMagazin := Sensor_CraneOnMagazin;
Crane.SliderMovedOut := Sensor_SliderMovedOut;
Crane.StartButtonMagazin := Sensor_StartButtonMagazin;
Actuator_CraneTurnCounterclockwise := Crane.CraneTurnCounterclockwise;
Actuator_CraneTurnClockwise := Crane.CraneTurnClockwise;
Actuator_CraneLower := Crane.CraneLower;
Actuator_MagazinVacuumOff := Crane.MagazinVacuumOff;
Actuator_MagazinVacuumOn := Crane.MagazinVacuumOn;
IF Sensor_MagazinEmergencyStop THEN
    Mag();
    Crane();
    IF Actuator_MagazinGreenLamp THEN
        IF (Crane.StartCommandCrane AND Mag.StartCommandMagazin) THEN
            Crane.StartVar := TRUE;
            Mag.StartVar := TRUE;
        END_IF;
    END_IF;
    Crane.SFCReset := FALSE;
    Mag.SFCReset := FALSE;
ELSIF NOT Sensor_MagazinEmergencyStop THEN
    Actuator_MagazinSlider := FALSE;
    Actuator_CraneLower := FALSE;
    Actuator_MagazinVacuumOn := FALSE;
    Actuator_MagazinVacuumOff := TRUE;
    Actuator_MagazinGreenLamp := FALSE;
    Actuator_CraneTurnCounterclockwise := FALSE;
    Actuator_CraneTurnClockwise := FALSE;
    Crane.SFCReset := TRUE;
    Mag.SFCReset := TRUE;
    Crane.StartVar := FALSE;
    Mag.StartVar := FALSE;
END_IF;
END_PROGRAM

CONFIGURATION Config0
  RESOURCE Res0 ON PLC
    TASK task0(INTERVAL := T#50ms, PRIORITY := 0);
    PROGRAM instance0 WITH task0 : Main;
  END_RESOURCE
END_CONFIGURATION

(* ---- Scenario0v0_Final.xml.st ---- *)
TYPE
    MAGAZIN_STATES_T : (GREEN_LAMP , INIT , INTERSTEP , MAGAZIN_INIT , MAGAZIN_INIT_2 , SLIDER_MOVE_BACK , START_MAGAZIN , STEP0 , STEP1 , CONVEY);
    CRANE_STATES_T : (CRANE_INIT , CRANE_INIT_2 , CRANE_LIFT_CONVEYOR , CRANE_LIFT_MAGAZINE , CRANE_ON_CONVEYOR , CRANE_STOP , CRANE_TURN_LEFT , INIT , INTERSTEP , INTERSTEP_2 , INTERSTEP_CHECK_WORKPIECE , MAGAZIN_STOP , START_CRANE , TIMEDELAY , TURN_RIGHT , RELEASE);
END_TYPE

FUNCTION_BLOCK MAGAZIN
    VAR_INPUT  CRANEDOWN : BOOL; END_VAR
    VAR_INPUT  CRANEONCONVEYOR : BOOL; END_VAR
    VAR_INPUT  CRANEONMAGAZIN : BOOL; END_VAR
    VAR_INPUT  CRANESUCKED : BOOL; END_VAR
    VAR_INPUT  CRANEUP : BOOL; END_VAR
    VAR_OUTPUT  MAGAZINGREENLAMP : BOOL; END_VAR
    VAR_OUTPUT  MAGAZINSLIDER : BOOL; END_VAR
    VAR  SFCINIT : BOOL; END_VAR
    VAR_INPUT  SFCRESET : BOOL; END_VAR
    VAR_INPUT  SLIDERMOVEDOUT : BOOL; END_VAR
    VAR_INPUT  SLIDERNOTMOVEDOUT : BOOL; END_VAR
    VAR_INPUT  STARTBUTTONMAGAZIN : BOOL; END_VAR
    VAR_OUTPUT  STARTCOMMANDMAGAZIN : BOOL; END_VAR
    VAR_INPUT  STARTVAR : BOOL; END_VAR
    VAR_INPUT  WORKPIECEREADY : BOOL; END_VAR
    VAR  _STATE : MAGAZIN_STATES_T; END_VAR
    VAR  _TRANSIT : BOOL; END_VAR
    VAR  INTERCONNECTMAGAZINESTARTCOMMAND : BOOL; END_VAR

    CASE _STATE OF
        MAGAZIN_STATES_T#GREEN_LAMP:
            _TRANSIT := FALSE;
            MAGAZINGREENLAMP := TRUE;
            INTERCONNECTMAGAZINESTARTCOMMAND := FALSE;
            IF TRUE THEN
                _TRANSIT := TRUE;
                _STATE := MAGAZIN_STATES_T#MAGAZIN_INIT;
            END_IF;

        MAGAZIN_STATES_T#INIT:
            _TRANSIT := FALSE;
            IF TRUE THEN
                _TRANSIT := TRUE;
                _STATE := MAGAZIN_STATES_T#START_MAGAZIN;
            END_IF;

        MAGAZIN_STATES_T#INTERSTEP:
            _TRANSIT := FALSE;
            STARTCOMMANDMAGAZIN := TRUE;
            IF STARTVAR THEN
                _TRANSIT := TRUE;
                _STATE := MAGAZIN_STATES_T#CONVEY;
            END_IF;

        MAGAZIN_STATES_T#MAGAZIN_INIT:
            _TRANSIT := FALSE;
            MAGAZINSLIDER := TRUE;
            IF TRUE THEN
                _TRANSIT := TRUE;
                _STATE := MAGAZIN_STATES_T#MAGAZIN_INIT_2;
            END_IF;

        MAGAZIN_STATES_T#MAGAZIN_INIT_2:
            _TRANSIT := FALSE;
            MAGAZINSLIDER := FALSE;
            IF TRUE THEN
                _TRANSIT := TRUE;
                _STATE := MAGAZIN_STATES_T#INTERSTEP;
            END_IF;

        MAGAZIN_STATES_T#SLIDER_MOVE_BACK:
            _TRANSIT := FALSE;
            IF ((SLIDERMOVEDOUT = TRUE) AND (SLIDERNOTMOVEDOUT = FALSE)) THEN
                MAGAZINSLIDER := FALSE;
            END_IF;
            IF CRANEUP THEN
                _TRANSIT := TRUE;
                _STATE := MAGAZIN_STATES_T#STEP1;
            END_IF;

        MAGAZIN_STATES_T#START_MAGAZIN:
            _TRANSIT := FALSE;
            MAGAZINSLIDER := FALSE;
            MAGAZINGREENLAMP := FALSE;
            STARTVAR := FALSE;
            STARTCOMMANDMAGAZIN := FALSE;
            IF (STARTBUTTONMAGAZIN = TRUE) THEN
                INTERCONNECTMAGAZINESTARTCOMMAND := TRUE;
            END_IF;
            IF INTERCONNECTMAGAZINESTARTCOMMAND THEN
                _TRANSIT := TRUE;
                _STATE := MAGAZIN_STATES_T#GREEN_LAMP;
            END_IF;

        MAGAZIN_STATES_T#STEP0:
            _TRANSIT := FALSE;
            IF CRANEDOWN THEN
                _TRANSIT := TRUE;
                _STATE := MAGAZIN_STATES_T#SLIDER_MOVE_BACK;
            END_IF;

        MAGAZIN_STATES_T#STEP1:
            _TRANSIT := FALSE;
            IF CRANEONCONVEYOR THEN
                _TRANSIT := TRUE;
                _STATE := MAGAZIN_STATES_T#INTERSTEP;
            END_IF;

        MAGAZIN_STATES_T#CONVEY:
            _TRANSIT := FALSE;
            IF SLIDERNOTMOVEDOUT THEN
                MAGAZINSLIDER := TRUE;
            END_IF;
            IF CRANEONMAGAZIN THEN
                _TRANSIT := TRUE;
                _STATE := MAGAZIN_STATES_T#STEP0;
            END_IF;

            END_CASE;
END_FUNCTION_BLOCK

FUNCTION_BLOCK CRANE_FB
    VAR_INPUT  CRANEDOWN : BOOL; END_VAR
    VAR_OUTPUT  CRANELOWER : BOOL; END_VAR
    VAR_INPUT  CRANEONCONVEYOR : BOOL; END_VAR
    VAR_INPUT  CRANEONMAGAZIN : BOOL; END_VAR
    VAR_INPUT  CRANESUCKED : BOOL; END_VAR
    VAR_OUTPUT  CRANETURNCLOCKWISE : BOOL; END_VAR
    VAR_OUTPUT  CRANETURNCOUNTERCLOCKWISE : BOOL; END_VAR
    VAR_INPUT  CRANEUP : BOOL; END_VAR
    VAR_OUTPUT  MAGAZINVACUUMOFF : BOOL; END_VAR
    VAR_OUTPUT  MAGAZINVACUUMON : BOOL; END_VAR
    VAR  SFCINIT : BOOL; END_VAR
    VAR_INPUT  SFCRESET : BOOL; END_VAR
    VAR_INPUT  SLIDERMOVEDOUT : BOOL; END_VAR
    VAR_INPUT  SLIDERNOTMOVEDOUT : BOOL; END_VAR
    VAR_INPUT  STARTBUTTONMAGAZIN : BOOL; END_VAR
    VAR_OUTPUT  STARTCOMMANDCRANE : BOOL; END_VAR
    VAR_INPUT  STARTVAR : BOOL; END_VAR
    VAR  TIMEDELAY_TIMER : TON; END_VAR
    VAR  TIMEDELAY_TIMER_DURATION : TIME := TIME#50MS; END_VAR
    VAR  TIMEDELAY_TIMER_INTERCONNECT : BOOL; END_VAR
    VAR_INPUT  WORKPIECEREADY : BOOL; END_VAR
    VAR  _STATE : CRANE_STATES_T; END_VAR
    VAR  _TRANSIT : BOOL; END_VAR
    VAR  INTERCONNECTCRANESTARTCOMMAND : BOOL; END_VAR

    CASE _STATE OF
        CRANE_STATES_T#CRANE_INIT:
            _TRANSIT := FALSE;
            CRANELOWER := TRUE;
            INTERCONNECTCRANESTARTCOMMAND := FALSE;
            IF CRANEDOWN THEN
                _TRANSIT := TRUE;
                _STATE := CRANE_STATES_T#CRANE_INIT_2;
            END_IF;

        CRANE_STATES_T#CRANE_INIT_2:
            _TRANSIT := FALSE;
            CRANELOWER := FALSE;
            IF CRANEUP THEN
                _TRANSIT := TRUE;
                _STATE := CRANE_STATES_T#INTERSTEP;
            END_IF;

        CRANE_STATES_T#CRANE_LIFT_CONVEYOR:
            _TRANSIT := FALSE;
            CRANELOWER := FALSE;
            IF TRUE THEN
                _TRANSIT := TRUE;
                _STATE := CRANE_STATES_T#INTERSTEP;
            END_IF;

        CRANE_STATES_T#CRANE_LIFT_MAGAZINE:
            _TRANSIT := FALSE;
            CRANELOWER := FALSE;
            IF CRANEUP THEN
                _TRANSIT := TRUE;
                _STATE := CRANE_STATES_T#CRANE_TURN_LEFT;
            END_IF;

        CRANE_STATES_T#CRANE_ON_CONVEYOR:
            _TRANSIT := FALSE;
            CRANETURNCOUNTERCLOCKWISE := FALSE;
            CRANETURNCLOCKWISE := FALSE;
            CRANELOWER := TRUE;
            IF CRANEDOWN THEN
                _TRANSIT := TRUE;
                _STATE := CRANE_STATES_T#RELEASE;
            END_IF;

        CRANE_STATES_T#CRANE_STOP:
            _TRANSIT := FALSE;
            IF TRUE THEN
                _TRANSIT := TRUE;
                _STATE := CRANE_STATES_T#START_CRANE;
            END_IF;

        CRANE_STATES_T#CRANE_TURN_LEFT:
            _TRANSIT := FALSE;
            CRANETURNCOUNTERCLOCKWISE := TRUE;
            CRANETURNCLOCKWISE := FALSE;
            IF CRANEONCONVEYOR THEN
                _TRANSIT := TRUE;
                _STATE := CRANE_STATES_T#CRANE_ON_CONVEYOR;
            END_IF;

        CRANE_STATES_T#INIT:
            _TRANSIT := FALSE;
            IF TRUE THEN
                _TRANSIT := TRUE;
                _STATE := CRANE_STATES_T#START_CRANE;
            END_IF;

        CRANE_STATES_T#INTERSTEP:
            _TRANSIT := FALSE;
            STARTCOMMANDCRANE := TRUE;
            IF STARTVAR THEN
                _TRANSIT := TRUE;
                _STATE := CRANE_STATES_T#INTERSTEP_2;
            END_IF;

        CRANE_STATES_T#INTERSTEP_2:
            _TRANSIT := FALSE;
            IF SLIDERMOVEDOUT THEN
                _TRANSIT := TRUE;
                _STATE := CRANE_STATES_T#TIMEDELAY;
            END_IF;

        CRANE_STATES_T#INTERSTEP_CHECK_WORKPIECE:
            _TRANSIT := FALSE;
            IF WORKPIECEREADY THEN
                _TRANSIT := TRUE;
                _STATE := CRANE_STATES_T#MAGAZIN_STOP;
            ELSIF NOT WORKPIECEREADY THEN
                _TRANSIT := TRUE;
                _STATE := CRANE_STATES_T#CRANE_STOP;
            END_IF;

        CRANE_STATES_T#MAGAZIN_STOP:
            _TRANSIT := FALSE;
            CRANETURNCLOCKWISE := FALSE;
            CRANETURNCOUNTERCLOCKWISE := FALSE;
            MAGAZINVACUUMON := TRUE;
            MAGAZINVACUUMOFF := FALSE;
            CRANELOWER := TRUE;
            IF CRANESUCKED THEN
                _TRANSIT := TRUE;
                _STATE := CRANE_STATES_T#CRANE_LIFT_MAGAZINE;
            END_IF;

        CRANE_STATES_T#START_CRANE:
            _TRANSIT := FALSE;
            CRANELOWER := FALSE;
            MAGAZINVACUUMOFF := TRUE;
            MAGAZINVACUUMON := FALSE;
            CRANETURNCOUNTERCLOCKWISE := FALSE;
            CRANETURNCLOCKWISE := FALSE;
            STARTVAR := FALSE;
            STARTCOMMANDCRANE := FALSE;
            IF (STARTBUTTONMAGAZIN = TRUE) THEN
                INTERCONNECTCRANESTARTCOMMAND := TRUE;
            END_IF;
            IF INTERCONNECTCRANESTARTCOMMAND THEN
                _TRANSIT := TRUE;
                _STATE := CRANE_STATES_T#CRANE_INIT;
            END_IF;

        CRANE_STATES_T#TIMEDELAY:
            _TRANSIT := FALSE;
            TIMEDELAY_TIMER(IN := TRUE, PT := TIMEDELAY_TIMER_DURATION);
            TIMEDELAY_TIMER_INTERCONNECT := TIMEDELAY_TIMER.Q;
            IF TIMEDELAY_TIMER_INTERCONNECT THEN
                _TRANSIT := TRUE;
                _STATE := CRANE_STATES_T#TURN_RIGHT;
            END_IF;

        CRANE_STATES_T#TURN_RIGHT:
            _TRANSIT := FALSE;
            CRANETURNCLOCKWISE := TRUE;
            CRANETURNCOUNTERCLOCKWISE := FALSE;
            IF CRANEONMAGAZIN THEN
                _TRANSIT := TRUE;
                _STATE := CRANE_STATES_T#INTERSTEP_CHECK_WORKPIECE;
            END_IF;

        CRANE_STATES_T#RELEASE:
            _TRANSIT := FALSE;
            MAGAZINVACUUMOFF := TRUE;
            MAGAZINVACUUMON := FALSE;
            IF TRUE THEN
                _TRANSIT := TRUE;
                _STATE := CRANE_STATES_T#CRANE_LIFT_CONVEYOR;
            END_IF;

            END_CASE;
END_FUNCTION_BLOCK

PROGRAM MAIN

VAR  ACTUATOR_CRANELOWER : BOOL; END_VAR
VAR  ACTUATOR_CRANETURNCLOCKWISE : BOOL; END_VAR
VAR  ACTUATOR_CRANETURNCOUNTERCLOCKWISE : BOOL; END_VAR
VAR  ACTUATOR_MAGAZINGREENLAMP : BOOL; END_VAR
VAR  ACTUATOR_MAGAZINSLIDER : BOOL; END_VAR
VAR  ACTUATOR_MAGAZINVACUUMOFF : BOOL; END_VAR
VAR  ACTUATOR_MAGAZINVACUUMON : BOOL; END_VAR
VAR  ACTUATOR_MAGAZINWHITELAMP : BOOL; END_VAR
VAR  CRANE : CRANE_FB; END_VAR
VAR  MAG : MAGAZIN; END_VAR
VAR  SENSOR_CRANEDOWN : BOOL; END_VAR
VAR  SENSOR_CRANEONCONVEYOR : BOOL; END_VAR
VAR  SENSOR_CRANEONMAGAZIN : BOOL; END_VAR
VAR  SENSOR_CRANEPOSITION : BOOL; END_VAR
VAR  SENSOR_CRANESUCKED : BOOL; END_VAR
VAR  SENSOR_CRANEUP : BOOL; END_VAR
VAR  SENSOR_MAGAZINEMERGENCYSTOP : BOOL; END_VAR
VAR  SENSOR_MAGAZINSWITCHMANUELLAUTOMATIC : BOOL; END_VAR
VAR  SENSOR_SLIDERMOVEDOUT : BOOL; END_VAR
VAR  SENSOR_SLIDERNOTMOVEDOUT : BOOL; END_VAR
VAR  SENSOR_STARTBUTTONMAGAZIN : BOOL; END_VAR
VAR  SENSOR_WORKPIECEREADY : BOOL; END_VAR
MAG.SLIDERNOTMOVEDOUT := SENSOR_SLIDERNOTMOVEDOUT;
MAG.SLIDERMOVEDOUT := SENSOR_SLIDERMOVEDOUT;
MAG.CRANEONMAGAZIN := SENSOR_CRANEONMAGAZIN;
MAG.CRANEDOWN := SENSOR_CRANEDOWN;
MAG.CRANEUP := SENSOR_CRANEUP;
MAG.CRANEONCONVEYOR := SENSOR_CRANEONCONVEYOR;
MAG.WORKPIECEREADY := SENSOR_WORKPIECEREADY;
MAG.STARTBUTTONMAGAZIN := SENSOR_STARTBUTTONMAGAZIN;
ACTUATOR_MAGAZINSLIDER := MAG.MAGAZINSLIDER;
ACTUATOR_MAGAZINGREENLAMP := MAG.MAGAZINGREENLAMP;
CRANE.WORKPIECEREADY := SENSOR_WORKPIECEREADY;
CRANE.CRANEUP := SENSOR_CRANEUP;
CRANE.CRANEONCONVEYOR := SENSOR_CRANEONCONVEYOR;
CRANE.CRANEDOWN := SENSOR_CRANEDOWN;
CRANE.CRANESUCKED := SENSOR_CRANESUCKED;
CRANE.CRANEONMAGAZIN := SENSOR_CRANEONMAGAZIN;
CRANE.SLIDERMOVEDOUT := SENSOR_SLIDERMOVEDOUT;
CRANE.STARTBUTTONMAGAZIN := SENSOR_STARTBUTTONMAGAZIN;
ACTUATOR_CRANETURNCOUNTERCLOCKWISE := CRANE.CRANETURNCOUNTERCLOCKWISE;
ACTUATOR_CRANETURNCLOCKWISE := CRANE.CRANETURNCLOCKWISE;
ACTUATOR_CRANELOWER := CRANE.CRANELOWER;
ACTUATOR_MAGAZINVACUUMOFF := CRANE.MAGAZINVACUUMOFF;
ACTUATOR_MAGAZINVACUUMON := CRANE.MAGAZINVACUUMON;
IF SENSOR_MAGAZINEMERGENCYSTOP THEN
    MAG();
    CRANE();
    IF ACTUATOR_MAGAZINGREENLAMP THEN
        IF (CRANE.STARTCOMMANDCRANE AND MAG.STARTCOMMANDMAGAZIN) THEN
            CRANE.STARTVAR := TRUE;
            MAG.STARTVAR := TRUE;
        END_IF;
    END_IF;
    CRANE.SFCRESET := FALSE;
    MAG.SFCRESET := FALSE;
ELSIF NOT SENSOR_MAGAZINEMERGENCYSTOP THEN
    ACTUATOR_MAGAZINSLIDER := FALSE;
    ACTUATOR_CRANELOWER := FALSE;
    ACTUATOR_MAGAZINVACUUMON := FALSE;
    ACTUATOR_MAGAZINVACUUMOFF := TRUE;
    ACTUATOR_MAGAZINGREENLAMP := FALSE;
    ACTUATOR_CRANETURNCOUNTERCLOCKWISE := FALSE;
    ACTUATOR_CRANETURNCLOCKWISE := FALSE;
    CRANE.SFCRESET := TRUE;
    MAG.SFCRESET := TRUE;
    CRANE.STARTVAR := FALSE;
    MAG.STARTVAR := FALSE;
END_IF;
END_PROGRAM

CONFIGURATION Config0
  RESOURCE Res0 ON PLC
    TASK TASK0(INTERVAL := T#50MS, PRIORITY := 0);
    PROGRAM INSTANCE0 WITH TASK0 : MAIN;
  END_RESOURCE
END_CONFIGURATION
